LIN {X 0,Y 468.404,Z 515.595,A -85,B 0,C 180,E1 -7638.313,E2 -7638.313} C_VEL
LIN {X 0,Y 467.88,Z 524.784,A -85,B 0,C 180,E1 -7639.397,E2 -7639.397} C_VEL
LIN {X 0,Y 467.447,Z 533.686,A -85,B 0,C 180,E1 -7640.699,E2 -7640.699} C_VEL
LIN {X 0,Y 467.093,Z 540.848,A -85,B 0,C 180,E1 -7642,E2 -7642} C_VEL
LIN {X 0,Y 466.908,Z 547.07,A -85,B 0,C 180,E1 -7643.438,E2 -7643.438} C_VEL
LIN {X 0,Y 466.784,Z 551.676,A -85,B 0,C 180,E1 -7644.817,E2 -7644.817} C_VEL
LIN {X 0,Y 466.663,Z 553.957,A -85,B 0,C 180,E1 -7645.681,E2 -7645.681} C_VEL
LIN {X 0,Y 466.695,Z 555.806,A -85,B 0,C 180,E1 -7646.547,E2 -7646.547} C_VEL
LIN {X 0,Y 466.646,Z 557.193,A -85,B 0,C 180,E1 -7647.41,E2 -7647.41} C_VEL
LIN {X 0,Y 466.589,Z 558.785,A -85,B 0,C 180,E1 -7649.137,E2 -7649.137} C_VEL
LIN {X 0,Y 466.57,Z 559,A -85,B 0,C 180,E1 -7650,E2 -7650} C_VEL
LIN {X 0,Y 466.589,Z 558.786,A -85,B 0,C 180,E1 -7650.863,E2 -7650.863} C_VEL
LIN {X 0,Y 466.646,Z 557.196,A -85,B 0,C 180,E1 -7652.59,E2 -7652.59} C_VEL
LIN {X 0,Y 466.695,Z 555.81,A -85,B 0,C 180,E1 -7653.453,E2 -7653.453} C_VEL
LIN {X 0,Y 466.703,Z 552.895,A -85,B 0,C 180,E1 -7654.751,E2 -7654.751} C_VEL
LIN {X 0,Y 466.839,Z 548.948,A -85,B 0,C 180,E1 -7656.049,E2 -7656.049} C_VEL
LIN {X 0,Y 466.998,Z 542.875,A -85,B 0,C 180,E1 -7657.567,E2 -7657.567} C_VEL
LIN {X 0,Y 467.35,Z 536.235,A -85,B 0,C 180,E1 -7658.867,E2 -7658.867} C_VEL
LIN {X 0,Y 467.737,Z 527.992,A -85,B 0,C 180,E1 -7660.169,E2 -7660.169} C_VEL
LIN {X 0,Y 468.135,Z 519.518,A -85,B 0,C 180,E1 -7661.254,E2 -7661.254} C_VEL
LIN {X 0,Y 468.687,Z 509.169,A -85,B 0,C 180,E1 -7662.321,E2 -7662.321} C_VEL
LIN {X 0,Y 469.111,Z 497.566,A -85,B 0,C 180,E1 -7663.284,E2 -7663.284} C_VEL
LIN {X 0,Y 469.632,Z 485.232,A -85,B 0,C 180,E1 -7664.074,E2 -7664.074} C_VEL
LIN {X 0,Y 470.084,Z 472.858,A -85,B 0,C 180,E1 -7664.668,E2 -7664.668} C_VEL
LIN {X 0,Y 469.97,Z 467.485,A -85,B 0,C 180,E1 -7664.88,E2 -7664.88} C_VEL
LIN {X 0,Y 467.715,Z 454.277,A -85,B 0,C 180,E1 -7665.333,E2 -7665.333} C_VEL
LIN {X 0,Y 467.222,Z 450.988,A -85,B 0,C 180,E1 -7665.43,E2 -7665.43} C_VEL
LIN {X 0,Y 467.484,Z 441.099,A -85,B 0,C 180,E1 -7668.715,E2 -7668.715} C_VEL
LIN {X 0,Y 467.721,Z 432.418,A -85,B 0,C 180,E1 -7671.634,E2 -7671.634} C_VEL
LIN {X 0,Y 468.026,Z 423.02,A -85,B 0,C 180,E1 -7674.863,E2 -7674.863} C_VEL
LIN {X 0,Y 468.406,Z 414.945,A -85,B 0,C 180,E1 -7677.719,E2 -7677.719} C_VEL
LIN {X 0,Y 468.801,Z 405.09,A -85,B 0,C 180,E1 -7681.294,E2 -7681.294} C_VEL
LIN {X 0,Y 469.172,Z 397.613,A -85,B 0,C 180,E1 -7684.097,E2 -7684.097} C_VEL
LIN {X 0,Y 469.316,Z 392.645,A -85,B 0,C 180,E1 -7686.036,E2 -7686.036} C_VEL
LIN {X 0,Y 468.318,Z 386.339,A -85,B 0,C 180,E1 -7688.706,E2 -7688.706} C_VEL
LIN {X 0,Y 467.58,Z 382.245,A -85,B 0,C 180,E1 -7690.618,E2 -7690.618} C_VEL
LIN {X 0,Y 467.57,Z 382.25,A -85,B 0,C 180,E1 -7693.823,E2 -7693.823} C_VEL
LIN {X 0,Y 467.559,Z 382.242,A -85,B 0,C 180,E1 -7696.256,E2 -7696.256} C_VEL
LIN {X 0,Y 467.581,Z 382.242,A -85,B 0,C 180,E1 -7698.723,E2 -7698.723} C_VEL
LIN {X 0,Y 467.569,Z 382.242,A -85,B 0,C 180,E1 -7701.956,E2 -7701.956} C_VEL
LIN {X 0,Y 467.57,Z 382.244,A -85,B 0,C 180,E1 -7705.168,E2 -7705.168} C_VEL
LIN {X 0,Y 467.586,Z 382.24,A -85,B 0,C 180,E1 -7708.26,E2 -7708.26} C_VEL
LIN {X 0,Y 467.58,Z 382.24,A -85,B 0,C 180,E1 -7711.251,E2 -7711.251} C_VEL
LIN {X 0,Y 467.616,Z 382.236,A -85,B 0,C 180,E1 -7713.2,E2 -7713.2} C_VEL
LIN {X 0,Y 467.594,Z 382.241,A -85,B 0,C 180,E1 -7716.469,E2 -7716.469} C_VEL
LIN {X 0,Y 467.628,Z 382.235,A -85,B 0,C 180,E1 -7719.777,E2 -7719.777} C_VEL
LIN {X 0,Y 467.613,Z 382.238,A -85,B 0,C 180,E1 -7722.507,E2 -7722.507} C_VEL
LIN {X 0,Y 467.61,Z 382.235,A -85,B 0,C 180,E1 -7725.197,E2 -7725.197} C_VEL
LIN {X 0,Y 467.687,Z 382.228,A -85,B 0,C 180,E1 -7727.855,E2 -7727.855} C_VEL
LIN {X 0,Y 467.686,Z 382.228,A -85,B 0,C 180,E1 -7731.357,E2 -7731.357} C_VEL
LIN {X 0,Y 467.747,Z 382.22,A -85,B 0,C 180,E1 -7733.963,E2 -7733.963} C_VEL
LIN {X 0,Y 467.863,Z 382.203,A -85,B 0,C 180,E1 -7737.417,E2 -7737.417} C_VEL
LIN {X 0,Y 467.887,Z 382.205,A -85,B 0,C 180,E1 -7740,E2 -7740} C_VEL
LIN {X 0,Y 467.862,Z 382.206,A -85,B 0,C 180,E1 -7742.583,E2 -7742.583} C_VEL
LIN {X 0,Y 467.748,Z 382.22,A -85,B 0,C 180,E1 -7746.037,E2 -7746.037} C_VEL
LIN {X 0,Y 467.683,Z 382.229,A -85,B 0,C 180,E1 -7748.643,E2 -7748.643} C_VEL
LIN {X 0,Y 467.66,Z 382.234,A -85,B 0,C 180,E1 -7752.145,E2 -7752.145} C_VEL
LIN {X 0,Y 467.643,Z 382.236,A -85,B 0,C 180,E1 -7755.695,E2 -7755.695} C_VEL
LIN {X 0,Y 467.627,Z 382.235,A -85,B 0,C 180,E1 -7759.308,E2 -7759.308} C_VEL
LIN {X 0,Y 467.538,Z 382.25,A -85,B 0,C 180,E1 -7762.074,E2 -7762.074} C_VEL
LIN {X 0,Y 467.589,Z 382.238,A -85,B 0,C 180,E1 -7764.888,E2 -7764.888} C_VEL
LIN {X 0,Y 467.631,Z 382.236,A -85,B 0,C 180,E1 -7767.768,E2 -7767.768} C_VEL
LIN {X 0,Y 467.571,Z 382.242,A -85,B 0,C 180,E1 -7771.045,E2 -7771.045} C_VEL
LIN {X 0,Y 467.592,Z 382.241,A -85,B 0,C 180,E1 -7774.242,E2 -7774.242} C_VEL
LIN {X 0,Y 467.551,Z 382.243,A -85,B 0,C 180,E1 -7777.186,E2 -7777.186} C_VEL
LIN {X 0,Y 467.581,Z 382.241,A -85,B 0,C 180,E1 -7780.265,E2 -7780.265} C_VEL
LIN {X 0,Y 467.589,Z 382.24,A -85,B 0,C 180,E1 -7782.567,E2 -7782.567} C_VEL
LIN {X 0,Y 467.575,Z 382.242,A -85,B 0,C 180,E1 -7786.177,E2 -7786.177} C_VEL
LIN {X 0,Y 467.587,Z 382.237,A -85,B 0,C 180,E1 -7788.722,E2 -7788.722} C_VEL
LIN {X 0,Y 467.564,Z 382.243,A -85,B 0,C 180,E1 -7791.955,E2 -7791.955} C_VEL
LIN {X 0,Y 467.434,Z 382.262,A -85,B 0,C 180,E1 -7795.156,E2 -7795.156} C_VEL
LIN {X 0,Y 467.22,Z 382.29,A -85,B 0,C 180,E1 -7797.391,E2 -7797.391} C_VEL
LIN {X 0,Y 467.124,Z 382.618,A -85,B 0,C 180,E1 -7798.225,E2 -7798.225} C_VEL
LIN {X 0,Y 467.082,Z 385.538,A -85,B 0,C 180,E1 -7801.217,E2 -7801.217} C_VEL
LIN {X 0,Y 467.017,Z 388.795,A -85,B 0,C 180,E1 -7804.545,E2 -7804.545} C_VEL
LIN {X 0,Y 466.878,Z 392.162,A -85,B 0,C 180,E1 -7807.893,E2 -7807.893} C_VEL
LIN {X 0,Y 466.856,Z 395.11,A -85,B 0,C 180,E1 -7810.659,E2 -7810.659} C_VEL
LIN {X 0,Y 466.821,Z 398.837,A -85,B 0,C 180,E1 -7813.93,E2 -7813.93} C_VEL
LIN {X 0,Y 466.77,Z 399.842,A -85,B 0,C 180,E1 -7814.23,E2 -7814.23} C_VEL
LIN {X 0,Y 466.543,Z 402.574,A -85,B 0,C 180,E1 -7814.555,E2 -7814.555} C_VEL
LIN {X 0,Y 466.119,Z 406.733,A -85,B 0,C 180,E1 -7814.803,E2 -7814.803} C_VEL
LIN {X 0,Y 463.509,Z 424.033,A -85,B 0,C 180,E1 -7815.447,E2 -7815.447} C_VEL
LIN {X 0,Y 463.214,Z 427.363,A -85,B 0,C 180,E1 -7815.614,E2 -7815.614} C_VEL
LIN {X 0,Y 462.772,Z 438.749,A -85,B 0,C 180,E1 -7816.313,E2 -7816.313} C_VEL
LIN {X 0,Y 462.312,Z 449.522,A -85,B 0,C 180,E1 -7817.154,E2 -7817.154} C_VEL
LIN {X 0,Y 461.81,Z 459.725,A -85,B 0,C 180,E1 -7818.144,E2 -7818.144} C_VEL
LIN {X 0,Y 461.272,Z 468.878,A -85,B 0,C 180,E1 -7819.243,E2 -7819.243} C_VEL
LIN {X 0,Y 460.84,Z 477.749,A -85,B 0,C 180,E1 -7820.564,E2 -7820.564} C_VEL
LIN {X 0,Y 460.394,Z 484.894,A -85,B 0,C 180,E1 -7821.883,E2 -7821.883} C_VEL
LIN {X 0,Y 460.123,Z 490.324,A -85,B 0,C 180,E1 -7823.133,E2 -7823.133} C_VEL
LIN {X 0,Y 459.892,Z 494.386,A -85,B 0,C 180,E1 -7824.299,E2 -7824.299} C_VEL
LIN {X 0,Y 459.881,Z 497.956,A -85,B 0,C 180,E1 -7825.618,E2 -7825.618} C_VEL
LIN {X 0,Y 459.779,Z 499.808,A -85,B 0,C 180,E1 -7826.495,E2 -7826.495} C_VEL
LIN {X 0,Y 459.768,Z 501.199,A -85,B 0,C 180,E1 -7827.372,E2 -7827.372} C_VEL
LIN {X 0,Y 459.557,Z 502.809,A -85,B 0,C 180,E1 -7829.124,E2 -7829.124} C_VEL
LIN {X 0,Y 459.536,Z 503.043,A -85,B 0,C 180,E1 -7830,E2 -7830} C_VEL
LIN {X 0,Y 459.639,Z 502.274,A -85,B 0,C 180,E1 -7831.753,E2 -7831.753} C_VEL
LIN {X 0,Y 459.768,Z 501.31,A -85,B 0,C 180,E1 -7832.628,E2 -7832.628} C_VEL
LIN {X 0,Y 459.78,Z 499.967,A -85,B 0,C 180,E1 -7833.505,E2 -7833.505} C_VEL
LIN {X 0,Y 459.846,Z 497.126,A -85,B 0,C 180,E1 -7834.822,E2 -7834.822} C_VEL
LIN {X 0,Y 460.021,Z 493.267,A -85,B 0,C 180,E1 -7836.139,E2 -7836.139} C_VEL
LIN {X 0,Y 460.196,Z 488.291,A -85,B 0,C 180,E1 -7837.459,E2 -7837.459} C_VEL
LIN {X 0,Y 460.571,Z 482.016,A -85,B 0,C 180,E1 -7838.777,E2 -7838.777} C_VEL
LIN {X 0,Y 460.971,Z 474.16,A -85,B 0,C 180,E1 -7840.098,E2 -7840.098} C_VEL
LIN {X 0,Y 461.518,Z 464.377,A -85,B 0,C 180,E1 -7841.418,E2 -7841.418} C_VEL
LIN {X 0,Y 462.073,Z 454.105,A -85,B 0,C 180,E1 -7842.518,E2 -7842.518} C_VEL
LIN {X 0,Y 462.528,Z 442.951,A -85,B 0,C 180,E1 -7843.476,E2 -7843.476} C_VEL
LIN {X 0,Y 463.071,Z 430.963,A -85,B 0,C 180,E1 -7844.278,E2 -7844.278} C_VEL
LIN {X 0,Y 463.458,Z 418.943,A -85,B 0,C 180,E1 -7844.883,E2 -7844.883} C_VEL
LIN {X 0,Y 463.495,Z 415.951,A -85,B 0,C 180,E1 -7845.012,E2 -7845.012} C_VEL
LIN {X 0,Y 460.557,Z 403.288,A -85,B 0,C 180,E1 -7845.535,E2 -7845.535} C_VEL
LIN {X 0,Y 459.806,Z 400.064,A -85,B 0,C 180,E1 -7845.667,E2 -7845.667} C_VEL
LIN {X 0,Y 459.784,Z 396.594,A -85,B 0,C 180,E1 -7848.723,E2 -7848.723} C_VEL
LIN {X 0,Y 459.828,Z 393.59,A -85,B 0,C 180,E1 -7851.52,E2 -7851.52} C_VEL
LIN {X 0,Y 459.896,Z 390.686,A -85,B 0,C 180,E1 -7854.369,E2 -7854.369} C_VEL
LIN {X 0,Y 459.989,Z 387.461,A -85,B 0,C 180,E1 -7857.605,E2 -7857.605} C_VEL
LIN {X 0,Y 460.056,Z 384.906,A -85,B 0,C 180,E1 -7860.273,E2 -7860.273} C_VEL
LIN {X 0,Y 460.108,Z 383.174,A -85,B 0,C 180,E1 -7862.318,E2 -7862.318} C_VEL
LIN {X 0,Y 460.434,Z 383.131,A -85,B 0,C 180,E1 -7865.453,E2 -7865.453} C_VEL
LIN {X 0,Y 460.548,Z 383.118,A -85,B 0,C 180,E1 -7868.898,E2 -7868.898} C_VEL
LIN {X 0,Y 460.527,Z 383.121,A -85,B 0,C 180,E1 -7872.181,E2 -7872.181} C_VEL
LIN {X 0,Y 460.517,Z 383.12,A -85,B 0,C 180,E1 -7875.411,E2 -7875.411} C_VEL
LIN {X 0,Y 460.536,Z 383.119,A -85,B 0,C 180,E1 -7878.398,E2 -7878.398} C_VEL
LIN {X 0,Y 460.531,Z 383.118,A -85,B 0,C 180,E1 -7881.267,E2 -7881.267} C_VEL
LIN {X 0,Y 460.517,Z 383.121,A -85,B 0,C 180,E1 -7884.555,E2 -7884.555} C_VEL
LIN {X 0,Y 460.536,Z 383.12,A -85,B 0,C 180,E1 -7887.716,E2 -7887.716} C_VEL
LIN {X 0,Y 460.545,Z 383.118,A -85,B 0,C 180,E1 -7890.769,E2 -7890.769} C_VEL
LIN {X 0,Y 460.56,Z 383.115,A -85,B 0,C 180,E1 -7893.734,E2 -7893.734} C_VEL
LIN {X 0,Y 460.549,Z 383.115,A -85,B 0,C 180,E1 -7896.624,E2 -7896.624} C_VEL
LIN {X 0,Y 460.557,Z 383.116,A -85,B 0,C 180,E1 -7899.453,E2 -7899.453} C_VEL
LIN {X 0,Y 460.555,Z 383.117,A -85,B 0,C 180,E1 -7902.23,E2 -7902.23} C_VEL
LIN {X 0,Y 460.571,Z 383.114,A -85,B 0,C 180,E1 -7904.965,E2 -7904.965} C_VEL
LIN {X 0,Y 460.616,Z 383.107,A -85,B 0,C 180,E1 -7908.559,E2 -7908.559} C_VEL
LIN {X 0,Y 460.625,Z 383.106,A -85,B 0,C 180,E1 -7911.224,E2 -7911.224} C_VEL
LIN {X 0,Y 460.712,Z 383.097,A -85,B 0,C 180,E1 -7913.87,E2 -7913.87} C_VEL
LIN {X 0,Y 460.804,Z 383.086,A -85,B 0,C 180,E1 -7917.377,E2 -7917.377} C_VEL
LIN {X 0,Y 460.858,Z 383.081,A -85,B 0,C 180,E1 -7920,E2 -7920} C_VEL
LIN {X 0,Y 460.805,Z 383.082,A -85,B 0,C 180,E1 -7922.622,E2 -7922.622} C_VEL
LIN {X 0,Y 460.715,Z 383.096,A -85,B 0,C 180,E1 -7926.13,E2 -7926.13} C_VEL
LIN {X 0,Y 460.634,Z 383.106,A -85,B 0,C 180,E1 -7928.776,E2 -7928.776} C_VEL
LIN {X 0,Y 460.639,Z 383.105,A -85,B 0,C 180,E1 -7932.457,E2 -7932.457} C_VEL
LIN {X 0,Y 460.605,Z 383.108,A -85,B 0,C 180,E1 -7935.997,E2 -7935.997} C_VEL
LIN {X 0,Y 460.574,Z 383.114,A -85,B 0,C 180,E1 -7939.615,E2 -7939.615} C_VEL
LIN {X 0,Y 460.515,Z 383.121,A -85,B 0,C 180,E1 -7942.428,E2 -7942.428} C_VEL
LIN {X 0,Y 460.557,Z 383.117,A -85,B 0,C 180,E1 -7945.798,E2 -7945.798} C_VEL
LIN {X 0,Y 460.56,Z 383.113,A -85,B 0,C 180,E1 -7948.233,E2 -7948.233} C_VEL
LIN {X 0,Y 460.525,Z 383.121,A -85,B 0,C 180,E1 -7951.283,E2 -7951.283} C_VEL
LIN {X 0,Y 460.536,Z 383.119,A -85,B 0,C 180,E1 -7954.505,E2 -7954.505} C_VEL
LIN {X 0,Y 460.505,Z 383.124,A -85,B 0,C 180,E1 -7957.623,E2 -7957.623} C_VEL
LIN {X 0,Y 460.545,Z 383.116,A -85,B 0,C 180,E1 -7960.269,E2 -7960.269} C_VEL
LIN {X 0,Y 460.504,Z 383.125,A -85,B 0,C 180,E1 -7963.375,E2 -7963.375} C_VEL
LIN {X 0,Y 460.512,Z 383.123,A -85,B 0,C 180,E1 -7966.626,E2 -7966.626} C_VEL
LIN {X 0,Y 460.571,Z 383.226,A -85,B 0,C 180,E1 -7969.188,E2 -7969.188} C_VEL
LIN {X 0,Y 461.891,Z 390.612,A -85,B 0,C 180,E1 -7972.509,E2 -7972.509} C_VEL
LIN {X 0,Y 462.366,Z 394.643,A -85,B 0,C 180,E1 -7974.206,E2 -7974.206} C_VEL
LIN {X 0,Y 461.99,Z 402.601,A -85,B 0,C 180,E1 -7977.313,E2 -7977.313} C_VEL
LIN {X 0,Y 461.572,Z 410.362,A -85,B 0,C 180,E1 -7980.215,E2 -7980.215} C_VEL
LIN {X 0,Y 461.217,Z 418.825,A -85,B 0,C 180,E1 -7983.287,E2 -7983.287} C_VEL
LIN {X 0,Y 460.863,Z 426.994,A -85,B 0,C 180,E1 -7986.203,E2 -7986.203} C_VEL
LIN {X 0,Y 460.613,Z 435.003,A -85,B 0,C 180,E1 -7988.994,E2 -7988.994} C_VEL
LIN {X 0,Y 460.37,Z 443.128,A -85,B 0,C 180,E1 -7991.763,E2 -7991.763} C_VEL
LIN {X 0,Y 460.167,Z 450.705,A -85,B 0,C 180,E1 -7994.337,E2 -7994.337} C_VEL
LIN {X 0,Y 462.581,Z 465.278,A -85,B 0,C 180,E1 -7994.812,E2 -7994.812} C_VEL
LIN {X 0,Y 463.264,Z 471.127,A -85,B 0,C 180,E1 -7995.054,E2 -7995.054} C_VEL
LIN {X 0,Y 462.835,Z 482.805,A -85,B 0,C 180,E1 -7995.602,E2 -7995.602} C_VEL
LIN {X 0,Y 462.286,Z 495.149,A -85,B 0,C 180,E1 -7996.37,E2 -7996.37} C_VEL
LIN {X 0,Y 461.877,Z 505.147,A -85,B 0,C 180,E1 -7997.162,E2 -7997.162} C_VEL
LIN {X 0,Y 461.399,Z 515.159,A -85,B 0,C 180,E1 -7998.133,E2 -7998.133} C_VEL
LIN {X 0,Y 460.865,Z 524.377,A -85,B 0,C 180,E1 -7999.233,E2 -7999.233} C_VEL
LIN {X 0,Y 460.418,Z 533.368,A -85,B 0,C 180,E1 -8000.555,E2 -8000.555} C_VEL
LIN {X 0,Y 460.055,Z 540.609,A -85,B 0,C 180,E1 -8001.876,E2 -8001.876} C_VEL
LIN {X 0,Y 459.848,Z 545.5,A -85,B 0,C 180,E1 -8002.977,E2 -8002.977} C_VEL
LIN {X 0,Y 459.756,Z 550.262,A -85,B 0,C 180,E1 -8004.297,E2 -8004.297} C_VEL
LIN {X 0,Y 459.579,Z 553.894,A -85,B 0,C 180,E1 -8005.615,E2 -8005.615} C_VEL
LIN {X 0,Y 459.591,Z 555.773,A -85,B 0,C 180,E1 -8006.493,E2 -8006.493} C_VEL
LIN {X 0,Y 459.57,Z 557.175,A -85,B 0,C 180,E1 -8007.37,E2 -8007.37} C_VEL
LIN {X 0,Y 459.494,Z 558.779,A -85,B 0,C 180,E1 -8009.124,E2 -8009.124} C_VEL
LIN {X 0,Y 459.474,Z 558.994,A -85,B 0,C 180,E1 -8010,E2 -8010} C_VEL
LIN {X 0,Y 459.494,Z 558.779,A -85,B 0,C 180,E1 -8010.876,E2 -8010.876} C_VEL
LIN {X 0,Y 459.57,Z 557.178,A -85,B 0,C 180,E1 -8012.629,E2 -8012.629} C_VEL
LIN {X 0,Y 459.591,Z 555.777,A -85,B 0,C 180,E1 -8013.507,E2 -8013.507} C_VEL
LIN {X 0,Y 459.634,Z 552.818,A -85,B 0,C 180,E1 -8014.824,E2 -8014.824} C_VEL
LIN {X 0,Y 459.757,Z 548.815,A -85,B 0,C 180,E1 -8016.143,E2 -8016.143} C_VEL
LIN {X 0,Y 459.929,Z 542.66,A -85,B 0,C 180,E1 -8017.684,E2 -8017.684} C_VEL
LIN {X 0,Y 460.287,Z 535.945,A -85,B 0,C 180,E1 -8019.004,E2 -8019.004} C_VEL
LIN {X 0,Y 460.7,Z 527.616,A -85,B 0,C 180,E1 -8020.326,E2 -8020.326} C_VEL
LIN {X 0,Y 461.146,Z 519.085,A -85,B 0,C 180,E1 -8021.427,E2 -8021.427} C_VEL
LIN {X 0,Y 461.697,Z 508.871,A -85,B 0,C 180,E1 -8022.498,E2 -8022.498} C_VEL
LIN {X 0,Y 462.119,Z 498.133,A -85,B 0,C 180,E1 -8023.41,E2 -8023.41} C_VEL
LIN {X 0,Y 462.643,Z 486.726,A -85,B 0,C 180,E1 -8024.179,E2 -8024.179} C_VEL
LIN {X 0,Y 463.147,Z 475.036,A -85,B 0,C 180,E1 -8024.781,E2 -8024.781} C_VEL
LIN {X 0,Y 463.102,Z 468.615,A -85,B 0,C 180,E1 -8025.048,E2 -8025.048} C_VEL
LIN {X 0,Y 460.884,Z 455.323,A -85,B 0,C 180,E1 -8025.529,E2 -8025.529} C_VEL
LIN {X 0,Y 460.148,Z 450.492,A -85,B 0,C 180,E1 -8025.689,E2 -8025.689} C_VEL
LIN {X 0,Y 460.454,Z 440.268,A -85,B 0,C 180,E1 -8029.178,E2 -8029.178} C_VEL
LIN {X 0,Y 460.728,Z 430.871,A -85,B 0,C 180,E1 -8032.418,E2 -8032.418} C_VEL
LIN {X 0,Y 461.117,Z 420.914,A -85,B 0,C 180,E1 -8035.942,E2 -8035.942} C_VEL
LIN {X 0,Y 461.43,Z 413.371,A -85,B 0,C 180,E1 -8038.671,E2 -8038.671} C_VEL
LIN {X 0,Y 461.828,Z 405.593,A -85,B 0,C 180,E1 -8041.548,E2 -8041.548} C_VEL
LIN {X 0,Y 462.191,Z 398.56,A -85,B 0,C 180,E1 -8044.237,E2 -8044.237} C_VEL
LIN {X 0,Y 462.263,Z 393.36,A -85,B 0,C 180,E1 -8046.314,E2 -8046.314} C_VEL
LIN {X 0,Y 461.257,Z 387.152,A -85,B 0,C 180,E1 -8049.007,E2 -8049.007} C_VEL
LIN {X 0,Y 460.553,Z 383.12,A -85,B 0,C 180,E1 -8050.911,E2 -8050.911} C_VEL
LIN {X 0,Y 460.522,Z 383.128,A -85,B 0,C 180,E1 -8054.171,E2 -8054.171} C_VEL
LIN {X 0,Y 460.516,Z 383.125,A -85,B 0,C 180,E1 -8057.1,E2 -8057.1} C_VEL
LIN {X 0,Y 460.561,Z 383.117,A -85,B 0,C 180,E1 -8060.14,E2 -8060.14} C_VEL
LIN {X 0,Y 460.481,Z 383.127,A -85,B 0,C 180,E1 -8063.471,E2 -8063.471} C_VEL
LIN {X 0,Y 460.532,Z 383.119,A -85,B 0,C 180,E1 -8066.675,E2 -8066.675} C_VEL
LIN {X 0,Y 460.514,Z 383.119,A -85,B 0,C 180,E1 -8069.76,E2 -8069.76} C_VEL
LIN {X 0,Y 460.581,Z 383.115,A -85,B 0,C 180,E1 -8072.757,E2 -8072.757} C_VEL
LIN {X 0,Y 460.534,Z 383.118,A -85,B 0,C 180,E1 -8075.667,E2 -8075.667} C_VEL
LIN {X 0,Y 460.525,Z 383.121,A -85,B 0,C 180,E1 -8078.578,E2 -8078.578} C_VEL
LIN {X 0,Y 460.595,Z 383.111,A -85,B 0,C 180,E1 -8081.311,E2 -8081.311} C_VEL
LIN {X 0,Y 460.607,Z 383.108,A -85,B 0,C 180,E1 -8084.059,E2 -8084.059} C_VEL
LIN {X 0,Y 460.634,Z 383.105,A -85,B 0,C 180,E1 -8087.667,E2 -8087.667} C_VEL
LIN {X 0,Y 460.633,Z 383.107,A -85,B 0,C 180,E1 -8091.224,E2 -8091.224} C_VEL
LIN {X 0,Y 460.713,Z 383.096,A -85,B 0,C 180,E1 -8093.87,E2 -8093.87} C_VEL
LIN {X 0,Y 460.804,Z 383.082,A -85,B 0,C 180,E1 -8097.378,E2 -8097.378} C_VEL
LIN {X 0,Y 460.857,Z 383.08,A -85,B 0,C 180,E1 -8100,E2 -8100} C_VEL
LIN {X 0,Y 460.803,Z 383.086,A -85,B 0,C 180,E1 -8102.623,E2 -8102.623} C_VEL
LIN {X 0,Y 460.714,Z 383.097,A -85,B 0,C 180,E1 -8106.13,E2 -8106.13} C_VEL
LIN {X 0,Y 460.631,Z 383.106,A -85,B 0,C 180,E1 -8108.776,E2 -8108.776} C_VEL
LIN {X 0,Y 460.617,Z 383.108,A -85,B 0,C 180,E1 -8112.445,E2 -8112.445} C_VEL
LIN {X 0,Y 460.604,Z 383.111,A -85,B 0,C 180,E1 -8115.998,E2 -8115.998} C_VEL
LIN {X 0,Y 460.573,Z 383.114,A -85,B 0,C 180,E1 -8119.615,E2 -8119.615} C_VEL
LIN {X 0,Y 460.514,Z 383.121,A -85,B 0,C 180,E1 -8122.429,E2 -8122.429} C_VEL
LIN {X 0,Y 460.556,Z 383.119,A -85,B 0,C 180,E1 -8125.798,E2 -8125.798} C_VEL
LIN {X 0,Y 460.559,Z 383.116,A -85,B 0,C 180,E1 -8128.233,E2 -8128.233} C_VEL
LIN {X 0,Y 460.524,Z 383.121,A -85,B 0,C 180,E1 -8131.283,E2 -8131.283} C_VEL
LIN {X 0,Y 460.535,Z 383.117,A -85,B 0,C 180,E1 -8134.506,E2 -8134.506} C_VEL
LIN {X 0,Y 460.531,Z 383.122,A -85,B 0,C 180,E1 -8137.621,E2 -8137.621} C_VEL
LIN {X 0,Y 460.545,Z 383.118,A -85,B 0,C 180,E1 -8140.269,E2 -8140.269} C_VEL
LIN {X 0,Y 460.499,Z 383.124,A -85,B 0,C 180,E1 -8143.376,E2 -8143.376} C_VEL
LIN {X 0,Y 460.526,Z 383.118,A -85,B 0,C 180,E1 -8146.627,E2 -8146.627} C_VEL
LIN {X 0,Y 460.546,Z 383.119,A -85,B 0,C 180,E1 -8149.73,E2 -8149.73} C_VEL
LIN {X 0,Y 460.498,Z 383.122,A -85,B 0,C 180,E1 -8152.525,E2 -8152.525} C_VEL
LIN {X 0,Y 460.357,Z 383.145,A -85,B 0,C 180,E1 -8155.608,E2 -8155.608} C_VEL
LIN {X 0,Y 460.117,Z 383.174,A -85,B 0,C 180,E1 -8157.683,E2 -8157.683} C_VEL
LIN {X 0,Y 460.04,Z 384.846,A -85,B 0,C 180,E1 -8159.726,E2 -8159.726} C_VEL
LIN {X 0,Y 459.98,Z 387.737,A -85,B 0,C 180,E1 -8162.718,E2 -8162.718} C_VEL
LIN {X 0,Y 459.905,Z 390.598,A -85,B 0,C 180,E1 -8165.632,E2 -8165.632} C_VEL
LIN {X 0,Y 459.821,Z 393.82,A -85,B 0,C 180,E1 -8168.803,E2 -8168.803} C_VEL
LIN {X 0,Y 459.792,Z 397.505,A -85,B 0,C 180,E1 -8172.199,E2 -8172.199} C_VEL
LIN {X 0,Y 459.796,Z 400.147,A -85,B 0,C 180,E1 -8174.45,E2 -8174.45} C_VEL
LIN {X 0,Y 462.964,Z 413.491,A -85,B 0,C 180,E1 -8174.968,E2 -8174.968} C_VEL
LIN {X 0,Y 463.514,Z 416.83,A -85,B 0,C 180,E1 -8175.119,E2 -8175.119} C_VEL
LIN {X 0,Y 463.214,Z 427.363,A -85,B 0,C 180,E1 -8175.614,E2 -8175.614} C_VEL
LIN {X 0,Y 462.367,Z 432.81,A -85,B 0,C 180,E1 -8175.903,E2 -8175.903} C_VEL
LIN {X 0,Y 459.267,Z 441.437,A -85,B 0,C 180,E1 -8176.384,E2 -8176.384} C_VEL
LIN {X 0,Y 456.107,Z 449.62,A -85,B 0,C 180,E1 -8176.948,E2 -8176.948} C_VEL
LIN {X 0,Y 455.164,Z 454.344,A -85,B 0,C 180,E1 -8177.363,E2 -8177.363} C_VEL
LIN {X 0,Y 454.589,Z 464.053,A -85,B 0,C 180,E1 -8178.406,E2 -8178.406} C_VEL
LIN {X 0,Y 454.142,Z 472.517,A -85,B 0,C 180,E1 -8179.523,E2 -8179.523} C_VEL
LIN {X 0,Y 453.677,Z 480.733,A -85,B 0,C 180,E1 -8180.864,E2 -8180.864} C_VEL
LIN {X 0,Y 453.339,Z 486.353,A -85,B 0,C 180,E1 -8181.98,E2 -8181.98} C_VEL
LIN {X 0,Y 453.083,Z 492.103,A -85,B 0,C 180,E1 -8183.398,E2 -8183.398} C_VEL
LIN {X 0,Y 452.724,Z 496.129,A -85,B 0,C 180,E1 -8184.656,E2 -8184.656} C_VEL
LIN {X 0,Y 452.809,Z 498.39,A -85,B 0,C 180,E1 -8185.549,E2 -8185.549} C_VEL
LIN {X 0,Y 452.718,Z 500.239,A -85,B 0,C 180,E1 -8186.44,E2 -8186.44} C_VEL
LIN {X 0,Y 452.697,Z 501.63,A -85,B 0,C 180,E1 -8187.331,E2 -8187.331} C_VEL
LIN {X 0,Y 452.493,Z 503.239,A -85,B 0,C 180,E1 -8189.11,E2 -8189.11} C_VEL
LIN {X 0,Y 452.47,Z 503.474,A -85,B 0,C 180,E1 -8190,E2 -8190} C_VEL
LIN {X 0,Y 452.58,Z 502.704,A -85,B 0,C 180,E1 -8191.78,E2 -8191.78} C_VEL
LIN {X 0,Y 452.683,Z 501.741,A -85,B 0,C 180,E1 -8192.67,E2 -8192.67} C_VEL
LIN {X 0,Y 452.718,Z 500.397,A -85,B 0,C 180,E1 -8193.56,E2 -8193.56} C_VEL
LIN {X 0,Y 452.772,Z 497.557,A -85,B 0,C 180,E1 -8194.898,E2 -8194.898} C_VEL
LIN {X 0,Y 452.986,Z 493.697,A -85,B 0,C 180,E1 -8196.235,E2 -8196.235} C_VEL
LIN {X 0,Y 453.163,Z 488.721,A -85,B 0,C 180,E1 -8197.575,E2 -8197.575} C_VEL
LIN {X 0,Y 453.556,Z 482.446,A -85,B 0,C 180,E1 -8198.914,E2 -8198.914} C_VEL
LIN {X 0,Y 454.007,Z 474.587,A -85,B 0,C 180,E1 -8200.255,E2 -8200.255} C_VEL
LIN {X 0,Y 454.572,Z 464.805,A -85,B 0,C 180,E1 -8201.595,E2 -8201.595} C_VEL
LIN {X 0,Y 455.175,Z 454.531,A -85,B 0,C 180,E1 -8202.711,E2 -8202.711} C_VEL
LIN {X 0,Y 455.637,Z 443.785,A -85,B 0,C 180,E1 -8203.651,E2 -8203.651} C_VEL
LIN {X 0,Y 456.131,Z 433.207,A -85,B 0,C 180,E1 -8204.386,E2 -8204.386} C_VEL
LIN {X 0,Y 456.573,Z 420.659,A -85,B 0,C 180,E1 -8205.056,E2 -8205.056} C_VEL
LIN {X 0,Y 456.552,Z 416.652,A -85,B 0,C 180,E1 -8205.233,E2 -8205.233} C_VEL
LIN {X 0,Y 453.59,Z 404.1,A -85,B 0,C 180,E1 -8205.77,E2 -8205.77} C_VEL
LIN {X 0,Y 452.716,Z 400.49,A -85,B 0,C 180,E1 -8205.905,E2 -8205.905} C_VEL
LIN {X 0,Y 452.711,Z 396.973,A -85,B 0,C 180,E1 -8209.027,E2 -8209.027} C_VEL
LIN {X 0,Y 452.769,Z 393.937,A -85,B 0,C 180,E1 -8211.872,E2 -8211.872} C_VEL
LIN {X 0,Y 452.86,Z 391.004,A -85,B 0,C 180,E1 -8214.773,E2 -8214.773} C_VEL
LIN {X 0,Y 452.935,Z 387.994,A -85,B 0,C 180,E1 -8217.816,E2 -8217.816} C_VEL
LIN {X 0,Y 452.992,Z 385.147,A -85,B 0,C 180,E1 -8220.796,E2 -8220.796} C_VEL
LIN {X 0,Y 453.008,Z 384.169,A -85,B 0,C 180,E1 -8221.836,E2 -8221.836} C_VEL
LIN {X 0,Y 453.364,Z 384.014,A -85,B 0,C 180,E1 -8225,E2 -8225} C_VEL
LIN {X 0,Y 453.466,Z 384,A -85,B 0,C 180,E1 -8228.312,E2 -8228.312} C_VEL
LIN {X 0,Y 453.498,Z 383.997,A -85,B 0,C 180,E1 -8230.609,E2 -8230.609} C_VEL
LIN {X 0,Y 453.458,Z 383.999,A -85,B 0,C 180,E1 -8233.244,E2 -8233.244} C_VEL
LIN {X 0,Y 453.466,Z 384,A -85,B 0,C 180,E1 -8235.779,E2 -8235.779} C_VEL
LIN {X 0,Y 453.483,Z 383.998,A -85,B 0,C 180,E1 -8238.209,E2 -8238.209} C_VEL
LIN {X 0,Y 453.52,Z 383.993,A -85,B 0,C 180,E1 -8240.79,E2 -8240.79} C_VEL
LIN {X 0,Y 453.461,Z 384,A -85,B 0,C 180,E1 -8243.918,E2 -8243.918} C_VEL
LIN {X 0,Y 453.487,Z 383.995,A -85,B 0,C 180,E1 -8247.151,E2 -8247.151} C_VEL
LIN {X 0,Y 453.48,Z 383.998,A -85,B 0,C 180,E1 -8250.268,E2 -8250.268} C_VEL
LIN {X 0,Y 453.506,Z 383.993,A -85,B 0,C 180,E1 -8253.294,E2 -8253.294} C_VEL
LIN {X 0,Y 453.503,Z 383.997,A -85,B 0,C 180,E1 -8256.239,E2 -8256.239} C_VEL
LIN {X 0,Y 453.488,Z 383.995,A -85,B 0,C 180,E1 -8259.118,E2 -8259.118} C_VEL
LIN {X 0,Y 453.509,Z 383.995,A -85,B 0,C 180,E1 -8261.944,E2 -8261.944} C_VEL
LIN {X 0,Y 453.545,Z 383.989,A -85,B 0,C 180,E1 -8264.726,E2 -8264.726} C_VEL
LIN {X 0,Y 453.564,Z 383.986,A -85,B 0,C 180,E1 -8268.379,E2 -8268.379} C_VEL
LIN {X 0,Y 453.59,Z 383.982,A -85,B 0,C 180,E1 -8271.087,E2 -8271.087} C_VEL
LIN {X 0,Y 453.678,Z 383.974,A -85,B 0,C 180,E1 -8273.775,E2 -8273.775} C_VEL
LIN {X 0,Y 453.748,Z 383.965,A -85,B 0,C 180,E1 -8277.337,E2 -8277.337} C_VEL
LIN {X 0,Y 453.828,Z 383.956,A -85,B 0,C 180,E1 -8280,E2 -8280} C_VEL
LIN {X 0,Y 453.749,Z 383.961,A -85,B 0,C 180,E1 -8282.663,E2 -8282.663} C_VEL
LIN {X 0,Y 453.682,Z 383.972,A -85,B 0,C 180,E1 -8286.225,E2 -8286.225} C_VEL
LIN {X 0,Y 453.598,Z 383.983,A -85,B 0,C 180,E1 -8288.913,E2 -8288.913} C_VEL
LIN {X 0,Y 453.607,Z 383.98,A -85,B 0,C 180,E1 -8292.551,E2 -8292.551} C_VEL
LIN {X 0,Y 453.549,Z 383.986,A -85,B 0,C 180,E1 -8296.196,E2 -8296.196} C_VEL
LIN {X 0,Y 453.523,Z 383.994,A -85,B 0,C 180,E1 -8299.04,E2 -8299.04} C_VEL
LIN {X 0,Y 453.481,Z 383.999,A -85,B 0,C 180,E1 -8301.836,E2 -8301.836} C_VEL
LIN {X 0,Y 453.505,Z 383.995,A -85,B 0,C 180,E1 -8304.735,E2 -8304.735} C_VEL
LIN {X 0,Y 453.542,Z 383.988,A -85,B 0,C 180,E1 -8307.961,E2 -8307.961} C_VEL
LIN {X 0,Y 453.47,Z 383.999,A -85,B 0,C 180,E1 -8311.525,E2 -8311.525} C_VEL
LIN {X 0,Y 453.491,Z 383.998,A -85,B 0,C 180,E1 -8314.777,E2 -8314.777} C_VEL
LIN {X 0,Y 453.468,Z 383.998,A -85,B 0,C 180,E1 -8318.311,E2 -8318.311} C_VEL
LIN {X 0,Y 453.497,Z 383.994,A -85,B 0,C 180,E1 -8320.609,E2 -8320.609} C_VEL
LIN {X 0,Y 453.46,Z 384.003,A -85,B 0,C 180,E1 -8323.244,E2 -8323.244} C_VEL
LIN {X 0,Y 453.477,Z 383.998,A -85,B 0,C 180,E1 -8325.78,E2 -8325.78} C_VEL
LIN {X 0,Y 453.541,Z 384.134,A -85,B 0,C 180,E1 -8328.89,E2 -8328.89} C_VEL
LIN {X 0,Y 454.948,Z 392.015,A -85,B 0,C 180,E1 -8332.496,E2 -8332.496} C_VEL
LIN {X 0,Y 455.374,Z 395.743,A -85,B 0,C 180,E1 -8334.093,E2 -8334.093} C_VEL
LIN {X 0,Y 455.093,Z 401.772,A -85,B 0,C 180,E1 -8336.504,E2 -8336.504} C_VEL
LIN {X 0,Y 454.698,Z 409.12,A -85,B 0,C 180,E1 -8339.332,E2 -8339.332} C_VEL
LIN {X 0,Y 454.269,Z 418.596,A -85,B 0,C 180,E1 -8342.845,E2 -8342.845} C_VEL
LIN {X 0,Y 453.792,Z 427.982,A -85,B 0,C 180,E1 -8346.255,E2 -8346.255} C_VEL
LIN {X 0,Y 453.541,Z 436.034,A -85,B 0,C 180,E1 -8349.12,E2 -8349.12} C_VEL
LIN {X 0,Y 453.258,Z 444.097,A -85,B 0,C 180,E1 -8351.934,E2 -8351.934} C_VEL
LIN {X 0,Y 453.085,Z 450.344,A -85,B 0,C 180,E1 -8354.094,E2 -8354.094} C_VEL
LIN {X 0,Y 455.398,Z 464.28,A -85,B 0,C 180,E1 -8354.547,E2 -8354.547} C_VEL
LIN {X 0,Y 456.337,Z 471.998,A -85,B 0,C 180,E1 -8354.879,E2 -8354.879} C_VEL
LIN {X 0,Y 455.831,Z 484.364,A -85,B 0,C 180,E1 -8355.49,E2 -8355.49} C_VEL
LIN {X 0,Y 455.292,Z 496.261,A -85,B 0,C 180,E1 -8356.271,E2 -8356.271} C_VEL
LIN {X 0,Y 454.808,Z 506.812,A -85,B 0,C 180,E1 -8357.154,E2 -8357.154} C_VEL
LIN {X 0,Y 454.294,Z 516.691,A -85,B 0,C 180,E1 -8358.172,E2 -8358.172} C_VEL
LIN {X 0,Y 453.73,Z 525.581,A -85,B 0,C 180,E1 -8359.288,E2 -8359.288} C_VEL
LIN {X 0,Y 453.31,Z 534.265,A -85,B 0,C 180,E1 -8360.631,E2 -8360.631} C_VEL
LIN {X 0,Y 452.924,Z 541.206,A -85,B 0,C 180,E1 -8361.972,E2 -8361.972} C_VEL
LIN {X 0,Y 452.73,Z 547.349,A -85,B 0,C 180,E1 -8363.47,E2 -8363.47} C_VEL
LIN {X 0,Y 452.567,Z 552.384,A -85,B 0,C 180,E1 -8365.1,E2 -8365.1} C_VEL
LIN {X 0,Y 452.494,Z 555.341,A -85,B 0,C 180,E1 -8366.438,E2 -8366.438} C_VEL
LIN {X 0,Y 452.496,Z 556.751,A -85,B 0,C 180,E1 -8367.329,E2 -8367.329} C_VEL
LIN {X 0,Y 452.433,Z 558.367,A -85,B 0,C 180,E1 -8369.11,E2 -8369.11} C_VEL
LIN {X 0,Y 452.41,Z 558.584,A -85,B 0,C 180,E1 -8370,E2 -8370} C_VEL
LIN {X 0,Y 452.433,Z 558.367,A -85,B 0,C 180,E1 -8370.89,E2 -8370.89} C_VEL
LIN {X 0,Y 452.496,Z 556.754,A -85,B 0,C 180,E1 -8372.671,E2 -8372.671} C_VEL
LIN {X 0,Y 452.494,Z 555.345,A -85,B 0,C 180,E1 -8373.562,E2 -8373.562} C_VEL
LIN {X 0,Y 452.567,Z 552.386,A -85,B 0,C 180,E1 -8374.9,E2 -8374.9} C_VEL
LIN {X 0,Y 452.691,Z 547.508,A -85,B 0,C 180,E1 -8376.486,E2 -8376.486} C_VEL
LIN {X 0,Y 452.926,Z 541.208,A -85,B 0,C 180,E1 -8378.028,E2 -8378.028} C_VEL
LIN {X 0,Y 453.31,Z 534.266,A -85,B 0,C 180,E1 -8379.369,E2 -8379.369} C_VEL
LIN {X 0,Y 453.728,Z 525.583,A -85,B 0,C 180,E1 -8380.712,E2 -8380.712} C_VEL
LIN {X 0,Y 454.294,Z 516.693,A -85,B 0,C 180,E1 -8381.828,E2 -8381.828} C_VEL
LIN {X 0,Y 454.795,Z 506.803,A -85,B 0,C 180,E1 -8382.847,E2 -8382.847} C_VEL
LIN {X 0,Y 455.259,Z 496.265,A -85,B 0,C 180,E1 -8383.73,E2 -8383.73} C_VEL
LIN {X 0,Y 455.825,Z 484.364,A -85,B 0,C 180,E1 -8384.51,E2 -8384.51} C_VEL
LIN {X 0,Y 456.346,Z 471.993,A -85,B 0,C 180,E1 -8385.12,E2 -8385.12} C_VEL
LIN {X 0,Y 454.857,Z 460.96,A -85,B 0,C 180,E1 -8385.575,E2 -8385.575} C_VEL
LIN {X 0,Y 453.105,Z 450.067,A -85,B 0,C 180,E1 -8385.933,E2 -8385.933} C_VEL
LIN {X 0,Y 453.363,Z 441.373,A -85,B 0,C 180,E1 -8388.998,E2 -8388.998} C_VEL
LIN {X 0,Y 453.606,Z 433.297,A -85,B 0,C 180,E1 -8391.83,E2 -8391.83} C_VEL
LIN {X 0,Y 453.98,Z 423.931,A -85,B 0,C 180,E1 -8395.197,E2 -8395.197} C_VEL
LIN {X 0,Y 454.38,Z 415.798,A -85,B 0,C 180,E1 -8398.16,E2 -8398.16} C_VEL
LIN {X 0,Y 454.857,Z 406.098,A -85,B 0,C 180,E1 -8401.809,E2 -8401.809} C_VEL
LIN {X 0,Y 455.27,Z 398.377,A -85,B 0,C 180,E1 -8404.832,E2 -8404.832} C_VEL
LIN {X 0,Y 455.217,Z 394.079,A -85,B 0,C 180,E1 -8406.6,E2 -8406.6} C_VEL
LIN {X 0,Y 454.173,Z 387.825,A -85,B 0,C 180,E1 -8409.379,E2 -8409.379} C_VEL
LIN {X 0,Y 453.506,Z 383.997,A -85,B 0,C 180,E1 -8411.195,E2 -8411.195} C_VEL
LIN {X 0,Y 453.494,Z 384.003,A -85,B 0,C 180,E1 -8414.53,E2 -8414.53} C_VEL
LIN {X 0,Y 453.481,Z 383.994,A -85,B 0,C 180,E1 -8418.209,E2 -8418.209} C_VEL
LIN {X 0,Y 453.518,Z 383.996,A -85,B 0,C 180,E1 -8420.79,E2 -8420.79} C_VEL
LIN {X 0,Y 453.459,Z 384,A -85,B 0,C 180,E1 -8423.917,E2 -8423.917} C_VEL
LIN {X 0,Y 453.486,Z 383.999,A -85,B 0,C 180,E1 -8427.151,E2 -8427.151} C_VEL
LIN {X 0,Y 453.478,Z 383.996,A -85,B 0,C 180,E1 -8430.268,E2 -8430.268} C_VEL
LIN {X 0,Y 453.508,Z 383.993,A -85,B 0,C 180,E1 -8433.294,E2 -8433.294} C_VEL
LIN {X 0,Y 453.501,Z 383.997,A -85,B 0,C 180,E1 -8436.239,E2 -8436.239} C_VEL
LIN {X 0,Y 453.487,Z 383.998,A -85,B 0,C 180,E1 -8439.118,E2 -8439.118} C_VEL
LIN {X 0,Y 453.516,Z 383.992,A -85,B 0,C 180,E1 -8441.945,E2 -8441.945} C_VEL
LIN {X 0,Y 453.544,Z 383.991,A -85,B 0,C 180,E1 -8444.726,E2 -8444.726} C_VEL
LIN {X 0,Y 453.606,Z 383.981,A -85,B 0,C 180,E1 -8447.472,E2 -8447.472} C_VEL
LIN {X 0,Y 453.597,Z 383.984,A -85,B 0,C 180,E1 -8451.087,E2 -8451.087} C_VEL
LIN {X 0,Y 453.681,Z 383.972,A -85,B 0,C 180,E1 -8453.775,E2 -8453.775} C_VEL
LIN {X 0,Y 453.748,Z 383.961,A -85,B 0,C 180,E1 -8457.337,E2 -8457.337} C_VEL
LIN {X 0,Y 453.828,Z 383.956,A -85,B 0,C 180,E1 -8460,E2 -8460} C_VEL
LIN {X 0,Y 453.747,Z 383.965,A -85,B 0,C 180,E1 -8462.663,E2 -8462.663} C_VEL
LIN {X 0,Y 453.681,Z 383.973,A -85,B 0,C 180,E1 -8466.225,E2 -8466.225} C_VEL
LIN {X 0,Y 453.594,Z 383.981,A -85,B 0,C 180,E1 -8468.913,E2 -8468.913} C_VEL
LIN {X 0,Y 453.567,Z 383.986,A -85,B 0,C 180,E1 -8472.529,E2 -8472.529} C_VEL
LIN {X 0,Y 453.548,Z 383.99,A -85,B 0,C 180,E1 -8476.196,E2 -8476.196} C_VEL
LIN {X 0,Y 453.521,Z 383.991,A -85,B 0,C 180,E1 -8479.04,E2 -8479.04} C_VEL
LIN {X 0,Y 453.48,Z 383.998,A -85,B 0,C 180,E1 -8481.836,E2 -8481.836} C_VEL
LIN {X 0,Y 453.504,Z 383.993,A -85,B 0,C 180,E1 -8484.735,E2 -8484.735} C_VEL
LIN {X 0,Y 453.541,Z 383.991,A -85,B 0,C 180,E1 -8487.961,E2 -8487.961} C_VEL
LIN {X 0,Y 453.469,Z 383.999,A -85,B 0,C 180,E1 -8491.525,E2 -8491.525} C_VEL
LIN {X 0,Y 453.49,Z 383.994,A -85,B 0,C 180,E1 -8494.777,E2 -8494.777} C_VEL
LIN {X 0,Y 453.476,Z 383.997,A -85,B 0,C 180,E1 -8498.311,E2 -8498.311} C_VEL
LIN {X 0,Y 453.497,Z 383.995,A -85,B 0,C 180,E1 -8500.609,E2 -8500.609} C_VEL
LIN {X 0,Y 453.456,Z 384.002,A -85,B 0,C 180,E1 -8503.244,E2 -8503.244} C_VEL
LIN {X 0,Y 453.478,Z 384,A -85,B 0,C 180,E1 -8505.78,E2 -8505.78} C_VEL
LIN {X 0,Y 453.497,Z 383.994,A -85,B 0,C 180,E1 -8508.211,E2 -8508.211} C_VEL
LIN {X 0,Y 453.497,Z 383.993,A -85,B 0,C 180,E1 -8510.793,E2 -8510.793} C_VEL
LIN {X 0,Y 453.414,Z 384.006,A -85,B 0,C 180,E1 -8513.913,E2 -8513.913} C_VEL
LIN {X 0,Y 453.172,Z 384.04,A -85,B 0,C 180,E1 -8516.873,E2 -8516.873} C_VEL
LIN {X 0,Y 453.008,Z 384.085,A -85,B 0,C 180,E1 -8518.165,E2 -8518.165} C_VEL
LIN {X 0,Y 452.945,Z 387.084,A -85,B 0,C 180,E1 -8521.249,E2 -8521.249} C_VEL
LIN {X 0,Y 452.876,Z 389.946,A -85,B 0,C 180,E1 -8524.245,E2 -8524.245} C_VEL
LIN {X 0,Y 452.778,Z 392.837,A -85,B 0,C 180,E1 -8527.167,E2 -8527.167} C_VEL
LIN {X 0,Y 452.722,Z 395.837,A -85,B 0,C 180,E1 -8530.03,E2 -8530.03} C_VEL
LIN {X 0,Y 452.709,Z 398.975,A -85,B 0,C 180,E1 -8532.845,E2 -8532.845} C_VEL
LIN {X 0,Y 452.726,Z 400.56,A -85,B 0,C 180,E1 -8534.195,E2 -8534.195} C_VEL
LIN {X 0,Y 456.085,Z 414.563,A -85,B 0,C 180,E1 -8534.76,E2 -8534.76} C_VEL
LIN {X 0,Y 456.64,Z 418.567,A -85,B 0,C 180,E1 -8534.947,E2 -8534.947} C_VEL
LIN {X 0,Y 456.274,Z 429.79,A -85,B 0,C 180,E1 -8535.505,E2 -8535.505} C_VEL
LIN {X 0,Y 455.815,Z 441.368,A -85,B 0,C 180,E1 -8536.257,E2 -8536.257} C_VEL
LIN {X 0,Y 455.291,Z 452.424,A -85,B 0,C 180,E1 -8537.18,E2 -8537.18} C_VEL
LIN {X 0,Y 455.164,Z 454.344,A -85,B 0,C 180,E1 -8537.363,E2 -8537.363} C_VEL
LIN {X 0,Y 454.197,Z 458.998,A -85,B 0,C 180,E1 -8537.808,E2 -8537.808} C_VEL
LIN {X 0,Y 450.923,Z 466.289,A -85,B 0,C 180,E1 -8538.557,E2 -8538.557} C_VEL
LIN {X 0,Y 447.753,Z 473.031,A -85,B 0,C 180,E1 -8539.39,E2 -8539.39} C_VEL
LIN {X 0,Y 446.955,Z 476.8,A -85,B 0,C 180,E1 -8539.961,E2 -8539.961} C_VEL
LIN {X 0,Y 446.437,Z 484.658,A -85,B 0,C 180,E1 -8541.399,E2 -8541.399} C_VEL
LIN {X 0,Y 446.098,Z 490.574,A -85,B 0,C 180,E1 -8542.76,E2 -8542.76} C_VEL
LIN {X 0,Y 445.817,Z 495.251,A -85,B 0,C 180,E1 -8544.119,E2 -8544.119} C_VEL
LIN {X 0,Y 445.739,Z 498.823,A -85,B 0,C 180,E1 -8545.478,E2 -8545.478} C_VEL
LIN {X 0,Y 445.658,Z 500.671,A -85,B 0,C 180,E1 -8546.383,E2 -8546.383} C_VEL
LIN {X 0,Y 445.615,Z 502.063,A -85,B 0,C 180,E1 -8547.288,E2 -8547.288} C_VEL
LIN {X 0,Y 445.43,Z 503.67,A -85,B 0,C 180,E1 -8549.096,E2 -8549.096} C_VEL
LIN {X 0,Y 445.405,Z 503.904,A -85,B 0,C 180,E1 -8550,E2 -8550} C_VEL
LIN {X 0,Y 445.523,Z 503.133,A -85,B 0,C 180,E1 -8551.808,E2 -8551.808} C_VEL
LIN {X 0,Y 445.603,Z 502.172,A -85,B 0,C 180,E1 -8552.712,E2 -8552.712} C_VEL
LIN {X 0,Y 445.658,Z 500.827,A -85,B 0,C 180,E1 -8553.617,E2 -8553.617} C_VEL
LIN {X 0,Y 445.706,Z 497.988,A -85,B 0,C 180,E1 -8554.975,E2 -8554.975} C_VEL
LIN {X 0,Y 445.954,Z 494.126,A -85,B 0,C 180,E1 -8556.334,E2 -8556.334} C_VEL
LIN {X 0,Y 446.154,Z 489.15,A -85,B 0,C 180,E1 -8557.695,E2 -8557.695} C_VEL
LIN {X 0,Y 446.557,Z 482.875,A -85,B 0,C 180,E1 -8559.055,E2 -8559.055} C_VEL
LIN {X 0,Y 447.049,Z 475.015,A -85,B 0,C 180,E1 -8560.416,E2 -8560.416} C_VEL
LIN {X 0,Y 447.63,Z 465.233,A -85,B 0,C 180,E1 -8561.777,E2 -8561.777} C_VEL
LIN {X 0,Y 448.286,Z 454.956,A -85,B 0,C 180,E1 -8562.909,E2 -8562.909} C_VEL
LIN {X 0,Y 448.806,Z 443.506,A -85,B 0,C 180,E1 -8563.92,E2 -8563.92} C_VEL
LIN {X 0,Y 449.387,Z 431.807,A -85,B 0,C 180,E1 -8564.723,E2 -8564.723} C_VEL
LIN {X 0,Y 449.798,Z 419.783,A -85,B 0,C 180,E1 -8565.346,E2 -8565.346} C_VEL
LIN {X 0,Y 449.536,Z 416.944,A -85,B 0,C 180,E1 -8565.483,E2 -8565.483} C_VEL
LIN {X 0,Y 446.438,Z 404.188,A -85,B 0,C 180,E1 -8566.039,E2 -8566.039} C_VEL
LIN {X 0,Y 445.685,Z 400.893,A -85,B 0,C 180,E1 -8566.17,E2 -8566.17} C_VEL
LIN {X 0,Y 445.635,Z 397.354,A -85,B 0,C 180,E1 -8569.341,E2 -8569.341} C_VEL
LIN {X 0,Y 445.707,Z 394.288,A -85,B 0,C 180,E1 -8572.237,E2 -8572.237} C_VEL
LIN {X 0,Y 445.787,Z 391.327,A -85,B 0,C 180,E1 -8575.193,E2 -8575.193} C_VEL
LIN {X 0,Y 445.871,Z 388.358,A -85,B 0,C 180,E1 -8578.221,E2 -8578.221} C_VEL
LIN {X 0,Y 445.974,Z 385.428,A -85,B 0,C 180,E1 -8581.335,E2 -8581.335} C_VEL
LIN {X 0,Y 446.043,Z 384.926,A -85,B 0,C 180,E1 -8582.393,E2 -8582.393} C_VEL
LIN {X 0,Y 446.343,Z 384.885,A -85,B 0,C 180,E1 -8585.633,E2 -8585.633} C_VEL
LIN {X 0,Y 446.447,Z 384.873,A -85,B 0,C 180,E1 -8589.027,E2 -8589.027} C_VEL
LIN {X 0,Y 446.438,Z 384.877,A -85,B 0,C 180,E1 -8592.277,E2 -8592.277} C_VEL
LIN {X 0,Y 446.455,Z 384.872,A -85,B 0,C 180,E1 -8595.104,E2 -8595.104} C_VEL
LIN {X 0,Y 446.432,Z 384.878,A -85,B 0,C 180,E1 -8598.609,E2 -8598.609} C_VEL
LIN {X 0,Y 446.465,Z 384.87,A -85,B 0,C 180,E1 -8600.975,E2 -8600.975} C_VEL
LIN {X 0,Y 446.425,Z 384.878,A -85,B 0,C 180,E1 -8604.374,E2 -8604.374} C_VEL
LIN {X 0,Y 446.427,Z 384.876,A -85,B 0,C 180,E1 -8607.639,E2 -8607.639} C_VEL
LIN {X 0,Y 446.453,Z 384.873,A -85,B 0,C 180,E1 -8610.791,E2 -8610.791} C_VEL
LIN {X 0,Y 446.482,Z 384.87,A -85,B 0,C 180,E1 -8613.849,E2 -8613.849} C_VEL
LIN {X 0,Y 446.431,Z 384.873,A -85,B 0,C 180,E1 -8616.823,E2 -8616.823} C_VEL
LIN {X 0,Y 446.449,Z 384.876,A -85,B 0,C 180,E1 -8619.737,E2 -8619.737} C_VEL
LIN {X 0,Y 446.462,Z 384.872,A -85,B 0,C 180,E1 -8622.597,E2 -8622.597} C_VEL
LIN {X 0,Y 446.475,Z 384.871,A -85,B 0,C 180,E1 -8625.412,E2 -8625.412} C_VEL
LIN {X 0,Y 446.522,Z 384.865,A -85,B 0,C 180,E1 -8628.193,E2 -8628.193} C_VEL
LIN {X 0,Y 446.537,Z 384.86,A -85,B 0,C 180,E1 -8630.945,E2 -8630.945} C_VEL
LIN {X 0,Y 446.646,Z 384.851,A -85,B 0,C 180,E1 -8633.676,E2 -8633.676} C_VEL
LIN {X 0,Y 446.695,Z 384.844,A -85,B 0,C 180,E1 -8637.295,E2 -8637.295} C_VEL
LIN {X 0,Y 446.798,Z 384.832,A -85,B 0,C 180,E1 -8640,E2 -8640} C_VEL
LIN {X 0,Y 446.696,Z 384.839,A -85,B 0,C 180,E1 -8642.705,E2 -8642.705} C_VEL
LIN {X 0,Y 446.652,Z 384.847,A -85,B 0,C 180,E1 -8646.324,E2 -8646.324} C_VEL
LIN {X 0,Y 446.544,Z 384.863,A -85,B 0,C 180,E1 -8649.055,E2 -8649.055} C_VEL
LIN {X 0,Y 446.539,Z 384.861,A -85,B 0,C 180,E1 -8652.729,E2 -8652.729} C_VEL
LIN {X 0,Y 446.493,Z 384.865,A -85,B 0,C 180,E1 -8656.459,E2 -8656.459} C_VEL
LIN {X 0,Y 446.473,Z 384.873,A -85,B 0,C 180,E1 -8659.303,E2 -8659.303} C_VEL
LIN {X 0,Y 446.422,Z 384.876,A -85,B 0,C 180,E1 -8662.199,E2 -8662.199} C_VEL
LIN {X 0,Y 446.448,Z 384.874,A -85,B 0,C 180,E1 -8665.153,E2 -8665.153} C_VEL
LIN {X 0,Y 446.489,Z 384.865,A -85,B 0,C 180,E1 -8668.178,E2 -8668.178} C_VEL
LIN {X 0,Y 446.423,Z 384.876,A -85,B 0,C 180,E1 -8671.775,E2 -8671.775} C_VEL
LIN {X 0,Y 446.433,Z 384.876,A -85,B 0,C 180,E1 -8674.523,E2 -8674.523} C_VEL
LIN {X 0,Y 446.419,Z 384.876,A -85,B 0,C 180,E1 -8678.079,E2 -8678.079} C_VEL
LIN {X 0,Y 446.431,Z 384.877,A -85,B 0,C 180,E1 -8680.917,E2 -8680.917} C_VEL
LIN {X 0,Y 446.405,Z 384.88,A -85,B 0,C 180,E1 -8683.846,E2 -8683.846} C_VEL
LIN {X 0,Y 446.424,Z 384.879,A -85,B 0,C 180,E1 -8686.4,E2 -8686.4} C_VEL
LIN {X 0,Y 446.461,Z 384.955,A -85,B 0,C 180,E1 -8688.537,E2 -8688.537} C_VEL
LIN {X 0,Y 447.68,Z 391.709,A -85,B 0,C 180,E1 -8691.715,E2 -8691.715} C_VEL
LIN {X 0,Y 448.41,Z 396.891,A -85,B 0,C 180,E1 -8694.003,E2 -8694.003} C_VEL
LIN {X 0,Y 448.078,Z 403.531,A -85,B 0,C 180,E1 -8696.704,E2 -8696.704} C_VEL
LIN {X 0,Y 447.594,Z 411.292,A -85,B 0,C 180,E1 -8699.723,E2 -8699.723} C_VEL
LIN {X 0,Y 447.211,Z 419.692,A -85,B 0,C 180,E1 -8702.887,E2 -8702.887} C_VEL
LIN {X 0,Y 446.744,Z 429.081,A -85,B 0,C 180,E1 -8706.349,E2 -8706.349} C_VEL
LIN {X 0,Y 446.449,Z 437.108,A -85,B 0,C 180,E1 -8709.256,E2 -8709.256} C_VEL
LIN {X 0,Y 446.164,Z 445.052,A -85,B 0,C 180,E1 -8712.111,E2 -8712.111} C_VEL
LIN {X 0,Y 446.004,Z 450.075,A -85,B 0,C 180,E1 -8713.844,E2 -8713.844} C_VEL
LIN {X 0,Y 448.18,Z 463.003,A -85,B 0,C 180,E1 -8714.265,E2 -8714.265} C_VEL
LIN {X 0,Y 449.414,Z 472.869,A -85,B 0,C 180,E1 -8714.699,E2 -8714.699} C_VEL
LIN {X 0,Y 448.959,Z 483.932,A -85,B 0,C 180,E1 -8715.263,E2 -8715.263} C_VEL
LIN {X 0,Y 448.36,Z 495.827,A -85,B 0,C 180,E1 -8716.054,E2 -8716.054} C_VEL
LIN {X 0,Y 447.819,Z 506.805,A -85,B 0,C 180,E1 -8716.992,E2 -8716.992} C_VEL
LIN {X 0,Y 447.321,Z 516.257,A -85,B 0,C 180,E1 -8717.984,E2 -8717.984} C_VEL
LIN {X 0,Y 446.703,Z 525.146,A -85,B 0,C 180,E1 -8719.117,E2 -8719.117} C_VEL
LIN {X 0,Y 446.259,Z 533.83,A -85,B 0,C 180,E1 -8720.482,E2 -8720.482} C_VEL
LIN {X 0,Y 445.884,Z 540.773,A -85,B 0,C 180,E1 -8721.845,E2 -8721.845} C_VEL
LIN {X 0,Y 445.65,Z 546.345,A -85,B 0,C 180,E1 -8723.208,E2 -8723.208} C_VEL
LIN {X 0,Y 445.541,Z 550.717,A -85,B 0,C 180,E1 -8724.569,E2 -8724.569} C_VEL
LIN {X 0,Y 445.427,Z 553.029,A -85,B 0,C 180,E1 -8725.475,E2 -8725.475} C_VEL
LIN {X 0,Y 445.398,Z 554.908,A -85,B 0,C 180,E1 -8726.381,E2 -8726.381} C_VEL
LIN {X 0,Y 445.423,Z 556.32,A -85,B 0,C 180,E1 -8727.287,E2 -8727.287} C_VEL
LIN {X 0,Y 445.372,Z 557.937,A -85,B 0,C 180,E1 -8729.096,E2 -8729.096} C_VEL
LIN {X 0,Y 445.349,Z 558.154,A -85,B 0,C 180,E1 -8730,E2 -8730} C_VEL
LIN {X 0,Y 445.372,Z 557.938,A -85,B 0,C 180,E1 -8730.904,E2 -8730.904} C_VEL
LIN {X 0,Y 445.423,Z 556.323,A -85,B 0,C 180,E1 -8732.713,E2 -8732.713} C_VEL
LIN {X 0,Y 445.398,Z 554.912,A -85,B 0,C 180,E1 -8733.619,E2 -8733.619} C_VEL
LIN {X 0,Y 445.5,Z 551.954,A -85,B 0,C 180,E1 -8734.977,E2 -8734.977} C_VEL
LIN {X 0,Y 445.587,Z 547.57,A -85,B 0,C 180,E1 -8736.451,E2 -8736.451} C_VEL
LIN {X 0,Y 445.804,Z 541.792,A -85,B 0,C 180,E1 -8737.929,E2 -8737.929} C_VEL
LIN {X 0,Y 446.186,Z 535.075,A -85,B 0,C 180,E1 -8739.291,E2 -8739.291} C_VEL
LIN {X 0,Y 446.628,Z 526.744,A -85,B 0,C 180,E1 -8740.655,E2 -8740.655} C_VEL
LIN {X 0,Y 447.187,Z 518.217,A -85,B 0,C 180,E1 -8741.789,E2 -8741.789} C_VEL
LIN {X 0,Y 447.72,Z 508.415,A -85,B 0,C 180,E1 -8742.854,E2 -8742.854} C_VEL
LIN {X 0,Y 448.263,Z 497.265,A -85,B 0,C 180,E1 -8743.833,E2 -8743.833} C_VEL
LIN {X 0,Y 448.831,Z 485.858,A -85,B 0,C 180,E1 -8744.625,E2 -8744.625} C_VEL
LIN {X 0,Y 449.385,Z 474.169,A -85,B 0,C 180,E1 -8745.244,E2 -8745.244} C_VEL
LIN {X 0,Y 449.224,Z 470.236,A -85,B 0,C 180,E1 -8745.424,E2 -8745.424} C_VEL
LIN {X 0,Y 447.139,Z 457.136,A -85,B 0,C 180,E1 -8745.95,E2 -8745.95} C_VEL
LIN {X 0,Y 446.007,Z 449.717,A -85,B 0,C 180,E1 -8746.182,E2 -8746.182} C_VEL
LIN {X 0,Y 446.327,Z 441.037,A -85,B 0,C 180,E1 -8749.31,E2 -8749.31} C_VEL
LIN {X 0,Y 446.642,Z 431.74,A -85,B 0,C 180,E1 -8752.676,E2 -8752.676} C_VEL
LIN {X 0,Y 447.083,Z 422.341,A -85,B 0,C 180,E1 -8756.114,E2 -8756.114} C_VEL
LIN {X 0,Y 447.422,Z 414.235,A -85,B 0,C 180,E1 -8759.14,E2 -8759.14} C_VEL
LIN {X 0,Y 447.917,Z 406.179,A -85,B 0,C 180,E1 -8762.241,E2 -8762.241} C_VEL
LIN {X 0,Y 448.37,Z 398.286,A -85,B 0,C 180,E1 -8765.405,E2 -8765.405} C_VEL
LIN {X 0,Y 448.187,Z 394.788,A -85,B 0,C 180,E1 -8766.895,E2 -8766.895} C_VEL
LIN {X 0,Y 446.986,Z 387.676,A -85,B 0,C 180,E1 -8770.139,E2 -8770.139} C_VEL
LIN {X 0,Y 446.456,Z 384.877,A -85,B 0,C 180,E1 -8771.539,E2 -8771.539} C_VEL
LIN {X 0,Y 446.457,Z 384.881,A -85,B 0,C 180,E1 -8775.103,E2 -8775.103} C_VEL
LIN {X 0,Y 446.43,Z 384.876,A -85,B 0,C 180,E1 -8778.609,E2 -8778.609} C_VEL
LIN {X 0,Y 446.464,Z 384.873,A -85,B 0,C 180,E1 -8780.975,E2 -8780.975} C_VEL
LIN {X 0,Y 446.424,Z 384.878,A -85,B 0,C 180,E1 -8784.374,E2 -8784.374} C_VEL
LIN {X 0,Y 446.425,Z 384.875,A -85,B 0,C 180,E1 -8787.639,E2 -8787.639} C_VEL
LIN {X 0,Y 446.452,Z 384.876,A -85,B 0,C 180,E1 -8790.791,E2 -8790.791} C_VEL
LIN {X 0,Y 446.481,Z 384.868,A -85,B 0,C 180,E1 -8793.849,E2 -8793.849} C_VEL
LIN {X 0,Y 446.429,Z 384.877,A -85,B 0,C 180,E1 -8796.823,E2 -8796.823} C_VEL
LIN {X 0,Y 446.448,Z 384.872,A -85,B 0,C 180,E1 -8799.737,E2 -8799.737} C_VEL
LIN {X 0,Y 446.468,Z 384.873,A -85,B 0,C 180,E1 -8802.597,E2 -8802.597} C_VEL
LIN {X 0,Y 446.474,Z 384.868,A -85,B 0,C 180,E1 -8805.413,E2 -8805.413} C_VEL
LIN {X 0,Y 446.543,Z 384.864,A -85,B 0,C 180,E1 -8808.194,E2 -8808.194} C_VEL
LIN {X 0,Y 446.604,Z 384.854,A -85,B 0,C 180,E1 -8811.858,E2 -8811.858} C_VEL
LIN {X 0,Y 446.649,Z 384.852,A -85,B 0,C 180,E1 -8814.583,E2 -8814.583} C_VEL
LIN {X 0,Y 446.668,Z 384.848,A -85,B 0,C 180,E1 -8818.197,E2 -8818.197} C_VEL
LIN {X 0,Y 446.798,Z 384.831,A -85,B 0,C 180,E1 -8820,E2 -8820} C_VEL
LIN {X 0,Y 446.694,Z 384.844,A -85,B 0,C 180,E1 -8822.705,E2 -8822.705} C_VEL
LIN {X 0,Y 446.651,Z 384.85,A -85,B 0,C 180,E1 -8826.324,E2 -8826.324} C_VEL
LIN {X 0,Y 446.54,Z 384.859,A -85,B 0,C 180,E1 -8829.055,E2 -8829.055} C_VEL
LIN {X 0,Y 446.525,Z 384.863,A -85,B 0,C 180,E1 -8832.73,E2 -8832.73} C_VEL
LIN {X 0,Y 446.499,Z 384.868,A -85,B 0,C 180,E1 -8836.228,E2 -8836.228} C_VEL
LIN {X 0,Y 446.472,Z 384.87,A -85,B 0,C 180,E1 -8839.303,E2 -8839.303} C_VEL
LIN {X 0,Y 446.422,Z 384.879,A -85,B 0,C 180,E1 -8842.2,E2 -8842.2} C_VEL
LIN {X 0,Y 446.447,Z 384.872,A -85,B 0,C 180,E1 -8845.153,E2 -8845.153} C_VEL
LIN {X 0,Y 446.488,Z 384.869,A -85,B 0,C 180,E1 -8848.179,E2 -8848.179} C_VEL
LIN {X 0,Y 446.422,Z 384.877,A -85,B 0,C 180,E1 -8851.775,E2 -8851.775} C_VEL
LIN {X 0,Y 446.432,Z 384.874,A -85,B 0,C 180,E1 -8854.523,E2 -8854.523} C_VEL
LIN {X 0,Y 446.433,Z 384.875,A -85,B 0,C 180,E1 -8858.082,E2 -8858.082} C_VEL
LIN {X 0,Y 446.43,Z 384.875,A -85,B 0,C 180,E1 -8860.918,E2 -8860.918} C_VEL
LIN {X 0,Y 446.401,Z 384.881,A -85,B 0,C 180,E1 -8863.846,E2 -8863.846} C_VEL
LIN {X 0,Y 446.449,Z 384.872,A -85,B 0,C 180,E1 -8866.397,E2 -8866.397} C_VEL
LIN {X 0,Y 446.446,Z 384.875,A -85,B 0,C 180,E1 -8869.802,E2 -8869.802} C_VEL
LIN {X 0,Y 446.409,Z 384.878,A -85,B 0,C 180,E1 -8872.121,E2 -8872.121} C_VEL
LIN {X 0,Y 446.319,Z 384.89,A -85,B 0,C 180,E1 -8874.967,E2 -8874.967} C_VEL
LIN {X 0,Y 445.959,Z 385.012,A -85,B 0,C 180,E1 -8878.321,E2 -8878.321} C_VEL
LIN {X 0,Y 445.871,Z 388.319,A -85,B 0,C 180,E1 -8881.779,E2 -8881.779} C_VEL
LIN {X 0,Y 445.795,Z 391.245,A -85,B 0,C 180,E1 -8884.808,E2 -8884.808} C_VEL
LIN {X 0,Y 445.71,Z 394.18,A -85,B 0,C 180,E1 -8887.763,E2 -8887.763} C_VEL
LIN {X 0,Y 445.704,Z 397.715,A -85,B 0,C 180,E1 -8891.103,E2 -8891.103} C_VEL
LIN {X 0,Y 445.688,Z 400.97,A -85,B 0,C 180,E1 -8893.942,E2 -8893.942} C_VEL
LIN {X 0,Y 448.916,Z 414.338,A -85,B 0,C 180,E1 -8894.484,E2 -8894.484} C_VEL
LIN {X 0,Y 449.817,Z 419.008,A -85,B 0,C 180,E1 -8894.713,E2 -8894.713} C_VEL
LIN {X 0,Y 449.44,Z 430.229,A -85,B 0,C 180,E1 -8895.279,E2 -8895.279} C_VEL
LIN {X 0,Y 448.94,Z 442.179,A -85,B 0,C 180,E1 -8896.071,E2 -8896.071} C_VEL
LIN {X 0,Y 448.402,Z 452.86,A -85,B 0,C 180,E1 -8896.979,E2 -8896.979} C_VEL
LIN {X 0,Y 447.864,Z 462.547,A -85,B 0,C 180,E1 -8897.999,E2 -8897.999} C_VEL
LIN {X 0,Y 447.265,Z 471.359,A -85,B 0,C 180,E1 -8899.131,E2 -8899.131} C_VEL
LIN {X 0,Y 446.955,Z 476.8,A -85,B 0,C 180,E1 -8899.961,E2 -8899.961} C_VEL
LIN {X 0,Y 446.144,Z 480.39,A -85,B 0,C 180,E1 -8900.555,E2 -8900.555} C_VEL
LIN {X 0,Y 442.942,Z 485.87,A -85,B 0,C 180,E1 -8901.539,E2 -8901.539} C_VEL
LIN {X 0,Y 439.749,Z 490.719,A -85,B 0,C 180,E1 -8902.586,E2 -8902.586} C_VEL
LIN {X 0,Y 438.965,Z 493.267,A -85,B 0,C 180,E1 -8903.272,E2 -8903.272} C_VEL
LIN {X 0,Y 438.629,Z 498.207,A -85,B 0,C 180,E1 -8904.944,E2 -8904.944} C_VEL
LIN {X 0,Y 438.599,Z 501.103,A -85,B 0,C 180,E1 -8906.325,E2 -8906.325} C_VEL
LIN {X 0,Y 438.537,Z 502.495,A -85,B 0,C 180,E1 -8907.244,E2 -8907.244} C_VEL
LIN {X 0,Y 438.37,Z 504.1,A -85,B 0,C 180,E1 -8909.081,E2 -8909.081} C_VEL
LIN {X 0,Y 438.343,Z 504.334,A -85,B 0,C 180,E1 -8910,E2 -8910} C_VEL
LIN {X 0,Y 438.468,Z 503.563,A -85,B 0,C 180,E1 -8911.837,E2 -8911.837} C_VEL
LIN {X 0,Y 438.599,Z 501.257,A -85,B 0,C 180,E1 -8913.675,E2 -8913.675} C_VEL
LIN {X 0,Y 438.627,Z 498.42,A -85,B 0,C 180,E1 -8915.056,E2 -8915.056} C_VEL
LIN {X 0,Y 438.914,Z 494.556,A -85,B 0,C 180,E1 -8916.436,E2 -8916.436} C_VEL
LIN {X 0,Y 439.125,Z 489.58,A -85,B 0,C 180,E1 -8917.819,E2 -8917.819} C_VEL
LIN {X 0,Y 439.567,Z 483.303,A -85,B 0,C 180,E1 -8919.2,E2 -8919.2} C_VEL
LIN {X 0,Y 440.084,Z 475.443,A -85,B 0,C 180,E1 -8920.583,E2 -8920.583} C_VEL
LIN {X 0,Y 440.694,Z 465.661,A -85,B 0,C 180,E1 -8921.965,E2 -8921.965} C_VEL
LIN {X 0,Y 441.402,Z 455.389,A -85,B 0,C 180,E1 -8923.113,E2 -8923.113} C_VEL
LIN {X 0,Y 441.942,Z 443.967,A -85,B 0,C 180,E1 -8924.138,E2 -8924.138} C_VEL
LIN {X 0,Y 442.543,Z 432.23,A -85,B 0,C 180,E1 -8924.955,E2 -8924.955} C_VEL
LIN {X 0,Y 442.988,Z 420.203,A -85,B 0,C 180,E1 -8925.588,E2 -8925.588} C_VEL
LIN {X 0,Y 440.53,Z 408.8,A -85,B 0,C 180,E1 -8926.132,E2 -8926.132} C_VEL
LIN {X 0,Y 438.601,Z 401.312,A -85,B 0,C 180,E1 -8926.436,E2 -8926.436} C_VEL
LIN {X 0,Y 438.588,Z 397.736,A -85,B 0,C 180,E1 -8929.664,E2 -8929.664} C_VEL
LIN {X 0,Y 438.647,Z 394.641,A -85,B 0,C 180,E1 -8932.615,E2 -8932.615} C_VEL
LIN {X 0,Y 438.725,Z 391.654,A -85,B 0,C 180,E1 -8935.628,E2 -8935.628} C_VEL
LIN {X 0,Y 438.803,Z 388.657,A -85,B 0,C 180,E1 -8938.718,E2 -8938.718} C_VEL
LIN {X 0,Y 438.95,Z 385.809,A -85,B 0,C 180,E1 -8941.942,E2 -8941.942} C_VEL
LIN {X 0,Y 439.305,Z 385.762,A -85,B 0,C 180,E1 -8945.323,E2 -8945.323} C_VEL
LIN {X 0,Y 439.381,Z 385.757,A -85,B 0,C 180,E1 -8948.596,E2 -8948.596} C_VEL
LIN {X 0,Y 439.392,Z 385.75,A -85,B 0,C 180,E1 -8951.257,E2 -8951.257} C_VEL
LIN {X 0,Y 439.403,Z 385.751,A -85,B 0,C 180,E1 -8954.73,E2 -8954.73} C_VEL
LIN {X 0,Y 439.399,Z 385.752,A -85,B 0,C 180,E1 -8957.796,E2 -8957.796} C_VEL
LIN {X 0,Y 439.441,Z 385.747,A -85,B 0,C 180,E1 -8960.229,E2 -8960.229} C_VEL
LIN {X 0,Y 439.381,Z 385.752,A -85,B 0,C 180,E1 -8963.713,E2 -8963.713} C_VEL
LIN {X 0,Y 439.376,Z 385.753,A -85,B 0,C 180,E1 -8967.054,E2 -8967.054} C_VEL
LIN {X 0,Y 439.387,Z 385.754,A -85,B 0,C 180,E1 -8970.274,E2 -8970.274} C_VEL
LIN {X 0,Y 439.432,Z 385.747,A -85,B 0,C 180,E1 -8973.396,E2 -8973.396} C_VEL
LIN {X 0,Y 439.389,Z 385.752,A -85,B 0,C 180,E1 -8976.43,E2 -8976.43} C_VEL
LIN {X 0,Y 439.393,Z 385.751,A -85,B 0,C 180,E1 -8979.397,E2 -8979.397} C_VEL
LIN {X 0,Y 439.431,Z 385.749,A -85,B 0,C 180,E1 -8982.309,E2 -8982.309} C_VEL
LIN {X 0,Y 439.453,Z 385.744,A -85,B 0,C 180,E1 -8985.174,E2 -8985.174} C_VEL
LIN {X 0,Y 439.488,Z 385.744,A -85,B 0,C 180,E1 -8988.001,E2 -8988.001} C_VEL
LIN {X 0,Y 439.509,Z 385.741,A -85,B 0,C 180,E1 -8991.725,E2 -8991.725} C_VEL
LIN {X 0,Y 439.624,Z 385.723,A -85,B 0,C 180,E1 -8994.496,E2 -8994.496} C_VEL
LIN {X 0,Y 439.639,Z 385.723,A -85,B 0,C 180,E1 -8998.168,E2 -8998.168} C_VEL
LIN {X 0,Y 439.767,Z 385.707,A -85,B 0,C 180,E1 -9000,E2 -9000} C_VEL
LIN {X 0,Y 439.645,Z 385.718,A -85,B 0,C 180,E1 -9002.749,E2 -9002.749} C_VEL
LIN {X 0,Y 439.623,Z 385.722,A -85,B 0,C 180,E1 -9006.425,E2 -9006.425} C_VEL
LIN {X 0,Y 439.506,Z 385.74,A -85,B 0,C 180,E1 -9009.201,E2 -9009.201} C_VEL
LIN {X 0,Y 439.509,Z 385.737,A -85,B 0,C 180,E1 -9012.726,E2 -9012.726} C_VEL
LIN {X 0,Y 439.451,Z 385.742,A -85,B 0,C 180,E1 -9016.348,E2 -9016.348} C_VEL
LIN {X 0,Y 439.407,Z 385.751,A -85,B 0,C 180,E1 -9019.626,E2 -9019.626} C_VEL
LIN {X 0,Y 439.368,Z 385.755,A -85,B 0,C 180,E1 -9022.575,E2 -9022.575} C_VEL
LIN {X 0,Y 439.402,Z 385.753,A -85,B 0,C 180,E1 -9025.585,E2 -9025.585} C_VEL
LIN {X 0,Y 439.422,Z 385.747,A -85,B 0,C 180,E1 -9028.673,E2 -9028.673} C_VEL
LIN {X 0,Y 439.374,Z 385.753,A -85,B 0,C 180,E1 -9032.03,E2 -9032.03} C_VEL
LIN {X 0,Y 439.398,Z 385.753,A -85,B 0,C 180,E1 -9035.34,E2 -9035.34} C_VEL
LIN {X 0,Y 439.387,Z 385.753,A -85,B 0,C 180,E1 -9038.595,E2 -9038.595} C_VEL
LIN {X 0,Y 439.392,Z 385.756,A -85,B 0,C 180,E1 -9041.257,E2 -9041.257} C_VEL
LIN {X 0,Y 439.406,Z 385.754,A -85,B 0,C 180,E1 -9044.729,E2 -9044.729} C_VEL
LIN {X 0,Y 439.424,Z 385.768,A -85,B 0,C 180,E1 -9048.172,E2 -9048.172} C_VEL
LIN {X 0,Y 440.62,Z 392.481,A -85,B 0,C 180,E1 -9051.404,E2 -9051.404} C_VEL
LIN {X 0,Y 441.445,Z 398.025,A -85,B 0,C 180,E1 -9053.909,E2 -9053.909} C_VEL
LIN {X 0,Y 441.092,Z 404.649,A -85,B 0,C 180,E1 -9056.654,E2 -9056.654} C_VEL
LIN {X 0,Y 440.617,Z 411.747,A -85,B 0,C 180,E1 -9059.465,E2 -9059.465} C_VEL
LIN {X 0,Y 440.242,Z 419.43,A -85,B 0,C 180,E1 -9062.422,E2 -9062.422} C_VEL
LIN {X 0,Y 439.814,Z 427.937,A -85,B 0,C 180,E1 -9065.621,E2 -9065.621} C_VEL
LIN {X 0,Y 439.419,Z 436.801,A -85,B 0,C 180,E1 -9068.908,E2 -9068.908} C_VEL
LIN {X 0,Y 439.12,Z 444.706,A -85,B 0,C 180,E1 -9071.814,E2 -9071.814} C_VEL
LIN {X 0,Y 438.972,Z 449.747,A -85,B 0,C 180,E1 -9073.58,E2 -9073.58} C_VEL
LIN {X 0,Y 441.122,Z 462.931,A -85,B 0,C 180,E1 -9074.019,E2 -9074.019} C_VEL
LIN {X 0,Y 442.533,Z 472.434,A -85,B 0,C 180,E1 -9074.455,E2 -9074.455} C_VEL
LIN {X 0,Y 442.095,Z 483.499,A -85,B 0,C 180,E1 -9075.029,E2 -9075.029} C_VEL
LIN {X 0,Y 441.438,Z 495.392,A -85,B 0,C 180,E1 -9075.831,E2 -9075.831} C_VEL
LIN {X 0,Y 440.82,Z 506.846,A -85,B 0,C 180,E1 -9076.829,E2 -9076.829} C_VEL
LIN {X 0,Y 440.217,Z 517.781,A -85,B 0,C 180,E1 -9078.021,E2 -9078.021} C_VEL
LIN {X 0,Y 439.612,Z 526.308,A -85,B 0,C 180,E1 -9079.173,E2 -9079.173} C_VEL
LIN {X 0,Y 439.152,Z 534.64,A -85,B 0,C 180,E1 -9080.559,E2 -9080.559} C_VEL
LIN {X 0,Y 438.752,Z 541.357,A -85,B 0,C 180,E1 -9081.943,E2 -9081.943} C_VEL
LIN {X 0,Y 438.546,Z 547.517,A -85,B 0,C 180,E1 -9083.559,E2 -9083.559} C_VEL
LIN {X 0,Y 438.434,Z 551.521,A -85,B 0,C 180,E1 -9084.942,E2 -9084.942} C_VEL
LIN {X 0,Y 438.303,Z 554.475,A -85,B 0,C 180,E1 -9086.323,E2 -9086.323} C_VEL
LIN {X 0,Y 438.351,Z 555.888,A -85,B 0,C 180,E1 -9087.243,E2 -9087.243} C_VEL
LIN {X 0,Y 438.283,Z 557.505,A -85,B 0,C 180,E1 -9089.081,E2 -9089.081} C_VEL
LIN {X 0,Y 438.29,Z 557.724,A -85,B 0,C 180,E1 -9090,E2 -9090} C_VEL
LIN {X 0,Y 438.283,Z 557.506,A -85,B 0,C 180,E1 -9090.919,E2 -9090.919} C_VEL
LIN {X 0,Y 438.351,Z 555.892,A -85,B 0,C 180,E1 -9092.757,E2 -9092.757} C_VEL
LIN {X 0,Y 438.303,Z 554.479,A -85,B 0,C 180,E1 -9093.677,E2 -9093.677} C_VEL
LIN {X 0,Y 438.434,Z 551.522,A -85,B 0,C 180,E1 -9095.058,E2 -9095.058} C_VEL
LIN {X 0,Y 438.506,Z 547.513,A -85,B 0,C 180,E1 -9096.442,E2 -9096.442} C_VEL
LIN {X 0,Y 438.753,Z 541.358,A -85,B 0,C 180,E1 -9098.057,E2 -9098.057} C_VEL
LIN {X 0,Y 439.152,Z 534.641,A -85,B 0,C 180,E1 -9099.441,E2 -9099.441} C_VEL
LIN {X 0,Y 439.611,Z 526.309,A -85,B 0,C 180,E1 -9100.827,E2 -9100.827} C_VEL
LIN {X 0,Y 440.212,Z 517.783,A -85,B 0,C 180,E1 -9101.979,E2 -9101.979} C_VEL
LIN {X 0,Y 440.745,Z 508.224,A -85,B 0,C 180,E1 -9103.037,E2 -9103.037} C_VEL
LIN {X 0,Y 441.332,Z 496.83,A -85,B 0,C 180,E1 -9104.055,E2 -9104.055} C_VEL
LIN {X 0,Y 441.956,Z 485.425,A -85,B 0,C 180,E1 -9104.858,E2 -9104.858} C_VEL
LIN {X 0,Y 442.508,Z 473.734,A -85,B 0,C 180,E1 -9105.487,E2 -9105.487} C_VEL
LIN {X 0,Y 441.052,Z 462.542,A -85,B 0,C 180,E1 -9105.996,E2 -9105.996} C_VEL
LIN {X 0,Y 438.957,Z 449.365,A -85,B 0,C 180,E1 -9106.452,E2 -9106.452} C_VEL
LIN {X 0,Y 439.258,Z 440.727,A -85,B 0,C 180,E1 -9109.633,E2 -9109.633} C_VEL
LIN {X 0,Y 439.636,Z 431.494,A -85,B 0,C 180,E1 -9113.058,E2 -9113.058} C_VEL
LIN {X 0,Y 440.085,Z 422.067,A -85,B 0,C 180,E1 -9116.561,E2 -9116.561} C_VEL
LIN {X 0,Y 440.387,Z 415.323,A -85,B 0,C 180,E1 -9119.126,E2 -9119.126} C_VEL
LIN {X 0,Y 440.919,Z 407.099,A -85,B 0,C 180,E1 -9122.35,E2 -9122.35} C_VEL
LIN {X 0,Y 441.331,Z 400.647,A -85,B 0,C 180,E1 -9124.98,E2 -9124.98} C_VEL
LIN {X 0,Y 441.284,Z 396.748,A -85,B 0,C 180,E1 -9126.641,E2 -9126.641} C_VEL
LIN {X 0,Y 440.405,Z 391.403,A -85,B 0,C 180,E1 -9129.088,E2 -9129.088} C_VEL
LIN {X 0,Y 439.404,Z 385.756,A -85,B 0,C 180,E1 -9131.829,E2 -9131.829} C_VEL
LIN {X 0,Y 439.405,Z 385.759,A -85,B 0,C 180,E1 -9135.271,E2 -9135.271} C_VEL
LIN {X 0,Y 439.391,Z 385.754,A -85,B 0,C 180,E1 -9138.743,E2 -9138.743} C_VEL
LIN {X 0,Y 439.388,Z 385.752,A -85,B 0,C 180,E1 -9141.606,E2 -9141.606} C_VEL
LIN {X 0,Y 439.403,Z 385.752,A -85,B 0,C 180,E1 -9144.844,E2 -9144.844} C_VEL
LIN {X 0,Y 439.376,Z 385.754,A -85,B 0,C 180,E1 -9148.14,E2 -9148.14} C_VEL
LIN {X 0,Y 439.435,Z 385.744,A -85,B 0,C 180,E1 -9151.598,E2 -9151.598} C_VEL
LIN {X 0,Y 439.401,Z 385.753,A -85,B 0,C 180,E1 -9154.415,E2 -9154.415} C_VEL
LIN {X 0,Y 439.367,Z 385.755,A -85,B 0,C 180,E1 -9157.425,E2 -9157.425} C_VEL
LIN {X 0,Y 439.445,Z 385.748,A -85,B 0,C 180,E1 -9160.663,E2 -9160.663} C_VEL
LIN {X 0,Y 439.466,Z 385.743,A -85,B 0,C 180,E1 -9164.225,E2 -9164.225} C_VEL
LIN {X 0,Y 439.511,Z 385.738,A -85,B 0,C 180,E1 -9168.002,E2 -9168.002} C_VEL
LIN {X 0,Y 439.552,Z 385.732,A -85,B 0,C 180,E1 -9171.726,E2 -9171.726} C_VEL
LIN {X 0,Y 439.624,Z 385.726,A -85,B 0,C 180,E1 -9174.496,E2 -9174.496} C_VEL
LIN {X 0,Y 439.638,Z 385.723,A -85,B 0,C 180,E1 -9178.168,E2 -9178.168} C_VEL
LIN {X 0,Y 439.768,Z 385.707,A -85,B 0,C 180,E1 -9180,E2 -9180} C_VEL
LIN {X 0,Y 439.643,Z 385.723,A -85,B 0,C 180,E1 -9182.749,E2 -9182.749} C_VEL
LIN {X 0,Y 439.622,Z 385.726,A -85,B 0,C 180,E1 -9186.425,E2 -9186.425} C_VEL
LIN {X 0,Y 439.502,Z 385.736,A -85,B 0,C 180,E1 -9189.202,E2 -9189.202} C_VEL
LIN {X 0,Y 439.469,Z 385.741,A -85,B 0,C 180,E1 -9192.938,E2 -9192.938} C_VEL
LIN {X 0,Y 439.45,Z 385.746,A -85,B 0,C 180,E1 -9196.348,E2 -9196.348} C_VEL
LIN {X 0,Y 439.406,Z 385.751,A -85,B 0,C 180,E1 -9199.626,E2 -9199.626} C_VEL
LIN {X 0,Y 439.368,Z 385.754,A -85,B 0,C 180,E1 -9202.575,E2 -9202.575} C_VEL
LIN {X 0,Y 439.401,Z 385.752,A -85,B 0,C 180,E1 -9205.585,E2 -9205.585} C_VEL
LIN {X 0,Y 439.421,Z 385.748,A -85,B 0,C 180,E1 -9208.673,E2 -9208.673} C_VEL
LIN {X 0,Y 439.374,Z 385.757,A -85,B 0,C 180,E1 -9212.031,E2 -9212.031} C_VEL
LIN {X 0,Y 439.397,Z 385.751,A -85,B 0,C 180,E1 -9215.34,E2 -9215.34} C_VEL
LIN {X 0,Y 439.393,Z 385.751,A -85,B 0,C 180,E1 -9218.594,E2 -9218.594} C_VEL
LIN {X 0,Y 439.391,Z 385.753,A -85,B 0,C 180,E1 -9221.257,E2 -9221.257} C_VEL
LIN {X 0,Y 439.403,Z 385.75,A -85,B 0,C 180,E1 -9224.729,E2 -9224.729} C_VEL
LIN {X 0,Y 439.414,Z 385.752,A -85,B 0,C 180,E1 -9227.798,E2 -9227.798} C_VEL
LIN {X 0,Y 439.428,Z 385.746,A -85,B 0,C 180,E1 -9230.227,E2 -9230.227} C_VEL
LIN {X 0,Y 439.319,Z 385.762,A -85,B 0,C 180,E1 -9233.707,E2 -9233.707} C_VEL
LIN {X 0,Y 439.12,Z 385.789,A -85,B 0,C 180,E1 -9236.331,E2 -9236.331} C_VEL
LIN {X 0,Y 438.938,Z 385.812,A -85,B 0,C 180,E1 -9238.104,E2 -9238.104} C_VEL
LIN {X 0,Y 438.801,Z 388.584,A -85,B 0,C 180,E1 -9241.282,E2 -9241.282} C_VEL
LIN {X 0,Y 438.741,Z 391.591,A -85,B 0,C 180,E1 -9244.374,E2 -9244.374} C_VEL
LIN {X 0,Y 438.649,Z 394.534,A -85,B 0,C 180,E1 -9247.386,E2 -9247.386} C_VEL
LIN {X 0,Y 438.659,Z 398.282,A -85,B 0,C 180,E1 -9250.957,E2 -9250.957} C_VEL
LIN {X 0,Y 438.629,Z 401.535,A -85,B 0,C 180,E1 -9253.679,E2 -9253.679} C_VEL
LIN {X 0,Y 441.917,Z 414.717,A -85,B 0,C 180,E1 -9254.229,E2 -9254.229} C_VEL
LIN {X 0,Y 442.948,Z 419.453,A -85,B 0,C 180,E1 -9254.47,E2 -9254.47} C_VEL
LIN {X 0,Y 442.607,Z 430.667,A -85,B 0,C 180,E1 -9255.047,E2 -9255.047} C_VEL
LIN {X 0,Y 442.092,Z 442.017,A -85,B 0,C 180,E1 -9255.805,E2 -9255.805} C_VEL
LIN {X 0,Y 441.519,Z 453.295,A -85,B 0,C 180,E1 -9256.773,E2 -9256.773} C_VEL
LIN {X 0,Y 440.934,Z 462.983,A -85,B 0,C 180,E1 -9257.808,E2 -9257.808} C_VEL
LIN {X 0,Y 440.325,Z 471.793,A -85,B 0,C 180,E1 -9258.958,E2 -9258.958} C_VEL
LIN {X 0,Y 439.804,Z 480.378,A -85,B 0,C 180,E1 -9260.341,E2 -9260.341} C_VEL
LIN {X 0,Y 439.307,Z 487.221,A -85,B 0,C 180,E1 -9261.722,E2 -9261.722} C_VEL
LIN {X 0,Y 438.965,Z 493.267,A -85,B 0,C 180,E1 -9263.272,E2 -9263.272} C_VEL
LIN {X 0,Y 438.22,Z 495.609,A -85,B 0,C 180,E1 -9263.975,E2 -9263.975} C_VEL
LIN {X 0,Y 435.195,Z 498.94,A -85,B 0,C 180,E1 -9265.134,E2 -9265.134} C_VEL
LIN {X 0,Y 432.658,Z 501.12,A -85,B 0,C 180,E1 -9266.09,E2 -9266.09} C_VEL
LIN {X 0,Y 431.56,Z 502.429,A -85,B 0,C 180,E1 -9266.843,E2 -9266.843} C_VEL
LIN {X 0,Y 431.466,Z 502.778,A -85,B 0,C 180,E1 -9267.099,E2 -9267.099} C_VEL
LIN {X 0,Y 431.384,Z 503.918,A -85,B 0,C 180,E1 -9268.133,E2 -9268.133} C_VEL
LIN {X 0,Y 431.282,Z 504.764,A -85,B 0,C 180,E1 -9270,E2 -9270} C_VEL
LIN {X 0,Y 431.312,Z 504.577,A -85,B 0,C 180,E1 -9270.934,E2 -9270.934} C_VEL
LIN {X 0,Y 431.453,Z 503.034,A -85,B 0,C 180,E1 -9272.801,E2 -9272.801} C_VEL
LIN {X 0,Y 431.543,Z 501.687,A -85,B 0,C 180,E1 -9273.735,E2 -9273.735} C_VEL
LIN {X 0,Y 431.553,Z 498.851,A -85,B 0,C 180,E1 -9275.139,E2 -9275.139} C_VEL
LIN {X 0,Y 431.875,Z 494.986,A -85,B 0,C 180,E1 -9276.541,E2 -9276.541} C_VEL
LIN {X 0,Y 432.119,Z 490.009,A -85,B 0,C 180,E1 -9277.946,E2 -9277.946} C_VEL
LIN {X 0,Y 432.588,Z 483.732,A -85,B 0,C 180,E1 -9279.35,E2 -9279.35} C_VEL
LIN {X 0,Y 433.129,Z 475.871,A -85,B 0,C 180,E1 -9280.755,E2 -9280.755} C_VEL
LIN {X 0,Y 433.769,Z 466.089,A -85,B 0,C 180,E1 -9282.159,E2 -9282.159} C_VEL
LIN {X 0,Y 434.517,Z 455.913,A -85,B 0,C 180,E1 -9283.315,E2 -9283.315} C_VEL
LIN {X 0,Y 435.05,Z 444.894,A -85,B 0,C 180,E1 -9284.324,E2 -9284.324} C_VEL
LIN {X 0,Y 435.604,Z 434.478,A -85,B 0,C 180,E1 -9285.08,E2 -9285.08} C_VEL
LIN {X 0,Y 436.134,Z 421.919,A -85,B 0,C 180,E1 -9285.779,E2 -9285.779} C_VEL
LIN {X 0,Y 435.166,Z 416.066,A -85,B 0,C 180,E1 -9286.08,E2 -9286.08} C_VEL
LIN {X 0,Y 431.829,Z 403.146,A -85,B 0,C 180,E1 -9286.648,E2 -9286.648} C_VEL
LIN {X 0,Y 431.558,Z 401.738,A -85,B 0,C 180,E1 -9286.701,E2 -9286.701} C_VEL
LIN {X 0,Y 431.536,Z 398.12,A -85,B 0,C 180,E1 -9289.999,E2 -9289.999} C_VEL
LIN {X 0,Y 431.6,Z 394.997,A -85,B 0,C 180,E1 -9293.005,E2 -9293.005} C_VEL
LIN {X 0,Y 431.711,Z 391.981,A -85,B 0,C 180,E1 -9296.075,E2 -9296.075} C_VEL
LIN {X 0,Y 431.782,Z 388.953,A -85,B 0,C 180,E1 -9299.229,E2 -9299.229} C_VEL
LIN {X 0,Y 431.856,Z 386.96,A -85,B 0,C 180,E1 -9301.384,E2 -9301.384} C_VEL
LIN {X 0,Y 432.122,Z 386.658,A -85,B 0,C 180,E1 -9303.956,E2 -9303.956} C_VEL
LIN {X 0,Y 432.299,Z 386.636,A -85,B 0,C 180,E1 -9306.979,E2 -9306.979} C_VEL
LIN {X 0,Y 432.337,Z 386.632,A -85,B 0,C 180,E1 -9310.179,E2 -9310.179} C_VEL
LIN {X 0,Y 432.32,Z 386.632,A -85,B 0,C 180,E1 -9313.061,E2 -9313.061} C_VEL
LIN {X 0,Y 432.336,Z 386.63,A -85,B 0,C 180,E1 -9315.665,E2 -9315.665} C_VEL
LIN {X 0,Y 432.336,Z 386.633,A -85,B 0,C 180,E1 -9318.398,E2 -9318.398} C_VEL
LIN {X 0,Y 432.351,Z 386.629,A -85,B 0,C 180,E1 -9321.851,E2 -9321.851} C_VEL
LIN {X 0,Y 432.345,Z 386.628,A -85,B 0,C 180,E1 -9325.323,E2 -9325.323} C_VEL
LIN {X 0,Y 432.326,Z 386.633,A -85,B 0,C 180,E1 -9328.654,E2 -9328.654} C_VEL
LIN {X 0,Y 432.386,Z 386.626,A -85,B 0,C 180,E1 -9331.877,E2 -9331.877} C_VEL
LIN {X 0,Y 432.351,Z 386.627,A -85,B 0,C 180,E1 -9334.999,E2 -9334.999} C_VEL
LIN {X 0,Y 432.362,Z 386.631,A -85,B 0,C 180,E1 -9338.046,E2 -9338.046} C_VEL
LIN {X 0,Y 432.389,Z 386.623,A -85,B 0,C 180,E1 -9341.03,E2 -9341.03} C_VEL
LIN {X 0,Y 432.435,Z 386.62,A -85,B 0,C 180,E1 -9343.961,E2 -9343.961} C_VEL
LIN {X 0,Y 432.464,Z 386.617,A -85,B 0,C 180,E1 -9347.803,E2 -9347.803} C_VEL
LIN {X 0,Y 432.469,Z 386.617,A -85,B 0,C 180,E1 -9351.59,E2 -9351.59} C_VEL
LIN {X 0,Y 432.601,Z 386.598,A -85,B 0,C 180,E1 -9354.406,E2 -9354.406} C_VEL
LIN {X 0,Y 432.608,Z 386.599,A -85,B 0,C 180,E1 -9358.138,E2 -9358.138} C_VEL
LIN {X 0,Y 432.737,Z 386.583,A -85,B 0,C 180,E1 -9360,E2 -9360} C_VEL
LIN {X 0,Y 432.597,Z 386.596,A -85,B 0,C 180,E1 -9362.794,E2 -9362.794} C_VEL
LIN {X 0,Y 432.578,Z 386.599,A -85,B 0,C 180,E1 -9366.53,E2 -9366.53} C_VEL
LIN {X 0,Y 432.449,Z 386.619,A -85,B 0,C 180,E1 -9369.353,E2 -9369.353} C_VEL
LIN {X 0,Y 432.45,Z 386.616,A -85,B 0,C 180,E1 -9372.812,E2 -9372.812} C_VEL
LIN {X 0,Y 432.416,Z 386.618,A -85,B 0,C 180,E1 -9376.478,E2 -9376.478} C_VEL
LIN {X 0,Y 432.343,Z 386.63,A -85,B 0,C 180,E1 -9379.96,E2 -9379.96} C_VEL
LIN {X 0,Y 432.322,Z 386.635,A -85,B 0,C 180,E1 -9382.964,E2 -9382.964} C_VEL
LIN {X 0,Y 432.365,Z 386.626,A -85,B 0,C 180,E1 -9386.032,E2 -9386.032} C_VEL
LIN {X 0,Y 432.347,Z 386.633,A -85,B 0,C 180,E1 -9389.187,E2 -9389.187} C_VEL
LIN {X 0,Y 432.327,Z 386.631,A -85,B 0,C 180,E1 -9392.443,E2 -9392.443} C_VEL
LIN {X 0,Y 432.348,Z 386.631,A -85,B 0,C 180,E1 -9395.632,E2 -9395.632} C_VEL
LIN {X 0,Y 432.354,Z 386.631,A -85,B 0,C 180,E1 -9399.342,E2 -9399.342} C_VEL
LIN {X 0,Y 432.337,Z 386.634,A -85,B 0,C 180,E1 -9401.797,E2 -9401.797} C_VEL
LIN {X 0,Y 432.337,Z 386.633,A -85,B 0,C 180,E1 -9404.347,E2 -9404.347} C_VEL
LIN {X 0,Y 432.375,Z 386.765,A -85,B 0,C 180,E1 -9407.894,E2 -9407.894} C_VEL
LIN {X 0,Y 433.419,Z 392.592,A -85,B 0,C 180,E1 -9410.773,E2 -9410.773} C_VEL
LIN {X 0,Y 434.332,Z 397.852,A -85,B 0,C 180,E1 -9413.222,E2 -9413.222} C_VEL
LIN {X 0,Y 434.349,Z 401.796,A -85,B 0,C 180,E1 -9414.941,E2 -9414.941} C_VEL
LIN {X 0,Y 433.833,Z 409.765,A -85,B 0,C 180,E1 -9418.231,E2 -9418.231} C_VEL
LIN {X 0,Y 433.289,Z 419.164,A -85,B 0,C 180,E1 -9421.94,E2 -9421.94} C_VEL
LIN {X 0,Y 432.779,Z 428.237,A -85,B 0,C 180,E1 -9425.422,E2 -9425.422} C_VEL
LIN {X 0,Y 432.321,Z 437.817,A -85,B 0,C 180,E1 -9429.044,E2 -9429.044} C_VEL
LIN {X 0,Y 431.997,Z 445.659,A -85,B 0,C 180,E1 -9431.995,E2 -9431.995} C_VEL
LIN {X 0,Y 431.869,Z 449.396,A -85,B 0,C 180,E1 -9433.304,E2 -9433.304} C_VEL
LIN {X 0,Y 434.063,Z 462.796,A -85,B 0,C 180,E1 -9433.763,E2 -9433.763} C_VEL
LIN {X 0,Y 435.639,Z 473.306,A -85,B 0,C 180,E1 -9434.262,E2 -9434.262} C_VEL
LIN {X 0,Y 435.091,Z 484.991,A -85,B 0,C 180,E1 -9434.902,E2 -9434.902} C_VEL
LIN {X 0,Y 434.425,Z 496.391,A -85,B 0,C 180,E1 -9435.717,E2 -9435.717} C_VEL
LIN {X 0,Y 433.804,Z 507.422,A -85,B 0,C 180,E1 -9436.714,E2 -9436.714} C_VEL
LIN {X 0,Y 433.231,Z 517.346,A -85,B 0,C 180,E1 -9437.825,E2 -9437.825} C_VEL
LIN {X 0,Y 432.576,Z 525.871,A -85,B 0,C 180,E1 -9438.994,E2 -9438.994} C_VEL
LIN {X 0,Y 432.103,Z 534.204,A -85,B 0,C 180,E1 -9440.403,E2 -9440.403} C_VEL
LIN {X 0,Y 431.711,Z 540.924,A -85,B 0,C 180,E1 -9441.811,E2 -9441.811} C_VEL
LIN {X 0,Y 431.459,Z 547.316,A -85,B 0,C 180,E1 -9443.528,E2 -9443.528} C_VEL
LIN {X 0,Y 431.369,Z 551.089,A -85,B 0,C 180,E1 -9444.859,E2 -9444.859} C_VEL
LIN {X 0,Y 431.21,Z 554.042,A -85,B 0,C 180,E1 -9446.262,E2 -9446.262} C_VEL
LIN {X 0,Y 431.28,Z 555.457,A -85,B 0,C 180,E1 -9447.198,E2 -9447.198} C_VEL
LIN {X 0,Y 431.198,Z 557.073,A -85,B 0,C 180,E1 -9449.066,E2 -9449.066} C_VEL
LIN {X 0,Y 431.216,Z 557.293,A -85,B 0,C 180,E1 -9450,E2 -9450} C_VEL
LIN {X 0,Y 431.198,Z 557.074,A -85,B 0,C 180,E1 -9450.934,E2 -9450.934} C_VEL
LIN {X 0,Y 431.28,Z 555.461,A -85,B 0,C 180,E1 -9452.802,E2 -9452.802} C_VEL
LIN {X 0,Y 431.21,Z 554.046,A -85,B 0,C 180,E1 -9453.738,E2 -9453.738} C_VEL
LIN {X 0,Y 431.369,Z 551.09,A -85,B 0,C 180,E1 -9455.141,E2 -9455.141} C_VEL
LIN {X 0,Y 431.441,Z 547.08,A -85,B 0,C 180,E1 -9456.547,E2 -9456.547} C_VEL
LIN {X 0,Y 431.712,Z 540.925,A -85,B 0,C 180,E1 -9458.189,E2 -9458.189} C_VEL
LIN {X 0,Y 432.103,Z 534.206,A -85,B 0,C 180,E1 -9459.597,E2 -9459.597} C_VEL
LIN {X 0,Y 432.574,Z 525.873,A -85,B 0,C 180,E1 -9461.005,E2 -9461.005} C_VEL
LIN {X 0,Y 433.221,Z 517.348,A -85,B 0,C 180,E1 -9462.175,E2 -9462.175} C_VEL
LIN {X 0,Y 433.806,Z 507.413,A -85,B 0,C 180,E1 -9463.287,E2 -9463.287} C_VEL
LIN {X 0,Y 434.412,Z 496.396,A -85,B 0,C 180,E1 -9464.283,E2 -9464.283} C_VEL
LIN {X 0,Y 435.076,Z 484.991,A -85,B 0,C 180,E1 -9465.098,E2 -9465.098} C_VEL
LIN {X 0,Y 435.607,Z 473.298,A -85,B 0,C 180,E1 -9465.739,E2 -9465.739} C_VEL
LIN {X 0,Y 433.58,Z 459.876,A -85,B 0,C 180,E1 -9466.351,E2 -9466.351} C_VEL
LIN {X 0,Y 431.871,Z 449.041,A -85,B 0,C 180,E1 -9466.721,E2 -9466.721} C_VEL
LIN {X 0,Y 432.209,Z 440.441,A -85,B 0,C 180,E1 -9469.967,E2 -9469.967} C_VEL
LIN {X 0,Y 432.556,Z 432.528,A -85,B 0,C 180,E1 -9472.951,E2 -9472.951} C_VEL
LIN {X 0,Y 433.03,Z 423.42,A -85,B 0,C 180,E1 -9476.396,E2 -9476.396} C_VEL
LIN {X 0,Y 433.36,Z 416.394,A -85,B 0,C 180,E1 -9479.112,E2 -9479.112} C_VEL
LIN {X 0,Y 433.896,Z 408.381,A -85,B 0,C 180,E1 -9482.311,E2 -9482.311} C_VEL
LIN {X 0,Y 434.35,Z 401.767,A -85,B 0,C 180,E1 -9485.058,E2 -9485.058} C_VEL
LIN {X 0,Y 434.285,Z 397.807,A -85,B 0,C 180,E1 -9486.782,E2 -9486.782} C_VEL
LIN {X 0,Y 433.236,Z 391.455,A -85,B 0,C 180,E1 -9489.758,E2 -9489.758} C_VEL
LIN {X 0,Y 432.375,Z 386.632,A -85,B 0,C 180,E1 -9492.262,E2 -9492.262} C_VEL
LIN {X 0,Y 432.335,Z 386.641,A -85,B 0,C 180,E1 -9495.665,E2 -9495.665} C_VEL
LIN {X 0,Y 432.335,Z 386.629,A -85,B 0,C 180,E1 -9498.398,E2 -9498.398} C_VEL
LIN {X 0,Y 432.35,Z 386.628,A -85,B 0,C 180,E1 -9501.851,E2 -9501.851} C_VEL
LIN {X 0,Y 432.343,Z 386.631,A -85,B 0,C 180,E1 -9505.323,E2 -9505.323} C_VEL
LIN {X 0,Y 432.324,Z 386.634,A -85,B 0,C 180,E1 -9508.654,E2 -9508.654} C_VEL
LIN {X 0,Y 432.385,Z 386.622,A -85,B 0,C 180,E1 -9511.877,E2 -9511.877} C_VEL
LIN {X 0,Y 432.349,Z 386.63,A -85,B 0,C 180,E1 -9514.999,E2 -9514.999} C_VEL
LIN {X 0,Y 432.36,Z 386.628,A -85,B 0,C 180,E1 -9518.046,E2 -9518.046} C_VEL
LIN {X 0,Y 432.39,Z 386.625,A -85,B 0,C 180,E1 -9521.03,E2 -9521.03} C_VEL
LIN {X 0,Y 432.434,Z 386.617,A -85,B 0,C 180,E1 -9523.961,E2 -9523.961} C_VEL
LIN {X 0,Y 432.484,Z 386.612,A -85,B 0,C 180,E1 -9527.804,E2 -9527.804} C_VEL
LIN {X 0,Y 432.496,Z 386.61,A -85,B 0,C 180,E1 -9531.59,E2 -9531.59} C_VEL
LIN {X 0,Y 432.601,Z 386.6,A -85,B 0,C 180,E1 -9534.406,E2 -9534.406} C_VEL
LIN {X 0,Y 432.608,Z 386.599,A -85,B 0,C 180,E1 -9538.138,E2 -9538.138} C_VEL
LIN {X 0,Y 432.738,Z 386.582,A -85,B 0,C 180,E1 -9540,E2 -9540} C_VEL
LIN {X 0,Y 432.595,Z 386.6,A -85,B 0,C 180,E1 -9542.794,E2 -9542.794} C_VEL
LIN {X 0,Y 432.577,Z 386.604,A -85,B 0,C 180,E1 -9546.53,E2 -9546.53} C_VEL
LIN {X 0,Y 432.445,Z 386.615,A -85,B 0,C 180,E1 -9549.353,E2 -9549.353} C_VEL
LIN {X 0,Y 432.434,Z 386.618,A -85,B 0,C 180,E1 -9552.804,E2 -9552.804} C_VEL
LIN {X 0,Y 432.415,Z 386.623,A -85,B 0,C 180,E1 -9556.479,E2 -9556.479} C_VEL
LIN {X 0,Y 432.342,Z 386.632,A -85,B 0,C 180,E1 -9559.96,E2 -9559.96} C_VEL
LIN {X 0,Y 432.321,Z 386.63,A -85,B 0,C 180,E1 -9562.964,E2 -9562.964} C_VEL
LIN {X 0,Y 432.364,Z 386.629,A -85,B 0,C 180,E1 -9566.033,E2 -9566.033} C_VEL
LIN {X 0,Y 432.346,Z 386.629,A -85,B 0,C 180,E1 -9569.187,E2 -9569.187} C_VEL
LIN {X 0,Y 432.326,Z 386.632,A -85,B 0,C 180,E1 -9572.443,E2 -9572.443} C_VEL
LIN {X 0,Y 432.347,Z 386.631,A -85,B 0,C 180,E1 -9575.632,E2 -9575.632} C_VEL
LIN {X 0,Y 432.355,Z 386.627,A -85,B 0,C 180,E1 -9578.717,E2 -9578.717} C_VEL
LIN {X 0,Y 432.336,Z 386.633,A -85,B 0,C 180,E1 -9581.797,E2 -9581.797} C_VEL
LIN {X 0,Y 432.381,Z 386.627,A -85,B 0,C 180,E1 -9585.659,E2 -9585.659} C_VEL
LIN {X 0,Y 432.371,Z 386.624,A -85,B 0,C 180,E1 -9588.393,E2 -9588.393} C_VEL
LIN {X 0,Y 432.337,Z 386.632,A -85,B 0,C 180,E1 -9591.85,E2 -9591.85} C_VEL
LIN {X 0,Y 432.195,Z 386.652,A -85,B 0,C 180,E1 -9595.309,E2 -9595.309} C_VEL
LIN {X 0,Y 431.831,Z 386.865,A -85,B 0,C 180,E1 -9598.614,E2 -9598.614} C_VEL
LIN {X 0,Y 431.768,Z 389.913,A -85,B 0,C 180,E1 -9601.833,E2 -9601.833} C_VEL
LIN {X 0,Y 431.668,Z 392.867,A -85,B 0,C 180,E1 -9604.956,E2 -9604.956} C_VEL
LIN {X 0,Y 431.585,Z 396.068,A -85,B 0,C 180,E1 -9608.156,E2 -9608.156} C_VEL
LIN {X 0,Y 431.596,Z 399.061,A -85,B 0,C 180,E1 -9610.993,E2 -9610.993} C_VEL
LIN {X 0,Y 431.565,Z 402.006,A -85,B 0,C 180,E1 -9613.404,E2 -9613.404} C_VEL
LIN {X 0,Y 434.954,Z 415.388,A -85,B 0,C 180,E1 -9613.978,E2 -9613.978} C_VEL
LIN {X 0,Y 436.143,Z 421.186,A -85,B 0,C 180,E1 -9614.281,E2 -9614.281} C_VEL
LIN {X 0,Y 435.698,Z 433.078,A -85,B 0,C 180,E1 -9614.924,E2 -9614.924} C_VEL
LIN {X 0,Y 435.176,Z 443.954,A -85,B 0,C 180,E1 -9615.695,E2 -9615.695} C_VEL
LIN {X 0,Y 434.564,Z 454.895,A -85,B 0,C 180,E1 -9616.676,E2 -9616.676} C_VEL
LIN {X 0,Y 433.8,Z 465.359,A -85,B 0,C 180,E1 -9617.842,E2 -9617.842} C_VEL
LIN {X 0,Y 433.26,Z 473.82,A -85,B 0,C 180,E1 -9619.012,E2 -9619.012} C_VEL
LIN {X 0,Y 432.712,Z 482.034,A -85,B 0,C 180,E1 -9620.417,E2 -9620.417} C_VEL
LIN {X 0,Y 432.288,Z 487.655,A -85,B 0,C 180,E1 -9621.586,E2 -9621.586} C_VEL
LIN {X 0,Y 431.927,Z 493.901,A -85,B 0,C 180,E1 -9623.221,E2 -9623.221} C_VEL
LIN {X 0,Y 431.556,Z 498.64,A -85,B 0,C 180,E1 -9624.861,E2 -9624.861} C_VEL
LIN {X 0,Y 431.543,Z 501.534,A -85,B 0,C 180,E1 -9626.265,E2 -9626.265} C_VEL
LIN {X 0,Y 431.466,Z 502.778,A -85,B 0,C 180,E1 -9627.099,E2 -9627.099} C_VEL
LIN {X 0,Y 430.764,Z 503.804,A -85,B 0,C 180,E1 -9627.866,E2 -9627.866} C_VEL
LIN {X 0,Y 427.822,Z 504.906,A -85,B 0,C 180,E1 -9629.122,E2 -9629.122} C_VEL
LIN {X 0,Y 425.358,Z 505.182,A -85,B 0,C 180,E1 -9630.141,E2 -9630.141} C_VEL
LIN {X 0,Y 424.318,Z 505.012,A -85,B 0,C 180,E1 -9630.929,E2 -9630.929} C_VEL
LIN {X 0,Y 424.244,Z 504.856,A -85,B 0,C 180,E1 -9631.196,E2 -9631.196} C_VEL
LIN {X 0,Y 424.384,Z 503.464,A -85,B 0,C 180,E1 -9632.848,E2 -9632.848} C_VEL
LIN {X 0,Y 424.487,Z 502.117,A -85,B 0,C 180,E1 -9633.797,E2 -9633.797} C_VEL
LIN {X 0,Y 424.484,Z 499.283,A -85,B 0,C 180,E1 -9635.225,E2 -9635.225} C_VEL
LIN {X 0,Y 424.835,Z 495.416,A -85,B 0,C 180,E1 -9636.65,E2 -9636.65} C_VEL
LIN {X 0,Y 425.094,Z 490.439,A -85,B 0,C 180,E1 -9638.079,E2 -9638.079} C_VEL
LIN {X 0,Y 425.589,Z 484.161,A -85,B 0,C 180,E1 -9639.505,E2 -9639.505} C_VEL
LIN {X 0,Y 426.173,Z 476.3,A -85,B 0,C 180,E1 -9640.932,E2 -9640.932} C_VEL
LIN {X 0,Y 426.737,Z 468.282,A -85,B 0,C 180,E1 -9642.121,E2 -9642.121} C_VEL
LIN {X 0,Y 427.47,Z 458.487,A -85,B 0,C 180,E1 -9643.307,E2 -9643.307} C_VEL
LIN {X 0,Y 428.026,Z 448.85,A -85,B 0,C 180,E1 -9644.258,E2 -9644.258} C_VEL
LIN {X 0,Y 428.619,Z 438.413,A -85,B 0,C 180,E1 -9645.088,E2 -9645.088} C_VEL
LIN {X 0,Y 429.178,Z 425.833,A -85,B 0,C 180,E1 -9645.859,E2 -9645.859} C_VEL
LIN {X 0,Y 429.129,Z 421.059,A -85,B 0,C 180,E1 -9646.105,E2 -9646.105} C_VEL
LIN {X 0,Y 426.189,Z 408.623,A -85,B 0,C 180,E1 -9646.726,E2 -9646.726} C_VEL
LIN {X 0,Y 424.481,Z 402.153,A -85,B 0,C 180,E1 -9646.992,E2 -9646.992} C_VEL
LIN {X 0,Y 424.477,Z 398.506,A -85,B 0,C 180,E1 -9650.347,E2 -9650.347} C_VEL
LIN {X 0,Y 424.55,Z 395.356,A -85,B 0,C 180,E1 -9653.41,E2 -9653.41} C_VEL
LIN {X 0,Y 424.649,Z 392.314,A -85,B 0,C 180,E1 -9656.542,E2 -9656.542} C_VEL
LIN {X 0,Y 424.749,Z 389.254,A -85,B 0,C 180,E1 -9659.762,E2 -9659.762} C_VEL
LIN {X 0,Y 424.845,Z 387.566,A -85,B 0,C 180,E1 -9661.963,E2 -9661.963} C_VEL
LIN {X 0,Y 425.205,Z 387.518,A -85,B 0,C 180,E1 -9665.345,E2 -9665.345} C_VEL
LIN {X 0,Y 425.279,Z 387.509,A -85,B 0,C 180,E1 -9667.695,E2 -9667.695} C_VEL
LIN {X 0,Y 425.283,Z 387.513,A -85,B 0,C 180,E1 -9670.52,E2 -9670.52} C_VEL
LIN {X 0,Y 425.261,Z 387.51,A -85,B 0,C 180,E1 -9673.351,E2 -9673.351} C_VEL
LIN {X 0,Y 425.261,Z 387.514,A -85,B 0,C 180,E1 -9676.649,E2 -9676.649} C_VEL
LIN {X 0,Y 425.299,Z 387.509,A -85,B 0,C 180,E1 -9679.874,E2 -9679.874} C_VEL
LIN {X 0,Y 425.289,Z 387.511,A -85,B 0,C 180,E1 -9682.487,E2 -9682.487} C_VEL
LIN {X 0,Y 425.312,Z 387.506,A -85,B 0,C 180,E1 -9685.818,E2 -9685.818} C_VEL
LIN {X 0,Y 425.295,Z 387.507,A -85,B 0,C 180,E1 -9689.239,E2 -9689.239} C_VEL
LIN {X 0,Y 425.353,Z 387.503,A -85,B 0,C 180,E1 -9692.442,E2 -9692.442} C_VEL
LIN {X 0,Y 425.352,Z 387.501,A -85,B 0,C 180,E1 -9695.602,E2 -9695.602} C_VEL
LIN {X 0,Y 425.298,Z 387.506,A -85,B 0,C 180,E1 -9698.682,E2 -9698.682} C_VEL
LIN {X 0,Y 425.335,Z 387.506,A -85,B 0,C 180,E1 -9701.703,E2 -9701.703} C_VEL
LIN {X 0,Y 425.353,Z 387.5,A -85,B 0,C 180,E1 -9704.671,E2 -9704.671} C_VEL
LIN {X 0,Y 425.417,Z 387.494,A -85,B 0,C 180,E1 -9707.598,E2 -9707.598} C_VEL
LIN {X 0,Y 425.413,Z 387.494,A -85,B 0,C 180,E1 -9711.449,E2 -9711.449} C_VEL
LIN {X 0,Y 425.556,Z 387.476,A -85,B 0,C 180,E1 -9714.313,E2 -9714.313} C_VEL
LIN {X 0,Y 425.578,Z 387.474,A -85,B 0,C 180,E1 -9718.107,E2 -9718.107} C_VEL
LIN {X 0,Y 425.707,Z 387.458,A -85,B 0,C 180,E1 -9720,E2 -9720} C_VEL
LIN {X 0,Y 425.55,Z 387.473,A -85,B 0,C 180,E1 -9722.84,E2 -9722.84} C_VEL
LIN {X 0,Y 425.536,Z 387.476,A -85,B 0,C 180,E1 -9726.639,E2 -9726.639} C_VEL
LIN {X 0,Y 425.408,Z 387.496,A -85,B 0,C 180,E1 -9729.509,E2 -9729.509} C_VEL
LIN {X 0,Y 425.409,Z 387.494,A -85,B 0,C 180,E1 -9732.91,E2 -9732.91} C_VEL
LIN {X 0,Y 425.365,Z 387.497,A -85,B 0,C 180,E1 -9736.605,E2 -9736.605} C_VEL
LIN {X 0,Y 425.333,Z 387.505,A -85,B 0,C 180,E1 -9739.636,E2 -9739.636} C_VEL
LIN {X 0,Y 425.309,Z 387.508,A -85,B 0,C 180,E1 -9743.365,E2 -9743.365} C_VEL
LIN {X 0,Y 425.352,Z 387.501,A -85,B 0,C 180,E1 -9746.844,E2 -9746.844} C_VEL
LIN {X 0,Y 425.295,Z 387.507,A -85,B 0,C 180,E1 -9749.719,E2 -9749.719} C_VEL
LIN {X 0,Y 425.286,Z 387.512,A -85,B 0,C 180,E1 -9753.048,E2 -9753.048} C_VEL
LIN {X 0,Y 425.287,Z 387.508,A -85,B 0,C 180,E1 -9755.929,E2 -9755.929} C_VEL
LIN {X 0,Y 425.301,Z 387.509,A -85,B 0,C 180,E1 -9759.043,E2 -9759.043} C_VEL
LIN {X 0,Y 425.278,Z 387.514,A -85,B 0,C 180,E1 -9762.653,E2 -9762.653} C_VEL
LIN {X 0,Y 425.272,Z 387.513,A -85,B 0,C 180,E1 -9766.045,E2 -9766.045} C_VEL
LIN {X 0,Y 425.35,Z 387.663,A -85,B 0,C 180,E1 -9767.56,E2 -9767.56} C_VEL
LIN {X 0,Y 426.491,Z 394.033,A -85,B 0,C 180,E1 -9770.76,E2 -9770.76} C_VEL
LIN {X 0,Y 427.322,Z 398.962,A -85,B 0,C 180,E1 -9773.109,E2 -9773.109} C_VEL
LIN {X 0,Y 427.38,Z 402.902,A -85,B 0,C 180,E1 -9774.861,E2 -9774.861} C_VEL
LIN {X 0,Y 426.836,Z 410.859,A -85,B 0,C 180,E1 -9778.204,E2 -9778.204} C_VEL
LIN {X 0,Y 426.245,Z 420.223,A -85,B 0,C 180,E1 -9781.971,E2 -9781.971} C_VEL
LIN {X 0,Y 425.696,Z 429.57,A -85,B 0,C 180,E1 -9785.623,E2 -9785.623} C_VEL
LIN {X 0,Y 425.237,Z 438.8,A -85,B 0,C 180,E1 -9789.186,E2 -9789.186} C_VEL
LIN {X 0,Y 424.896,Z 446.604,A -85,B 0,C 180,E1 -9792.181,E2 -9792.181} C_VEL
LIN {X 0,Y 424.79,Z 448.725,A -85,B 0,C 180,E1 -9792.993,E2 -9792.993} C_VEL
LIN {X 0,Y 427.268,Z 464.198,A -85,B 0,C 180,E1 -9793.569,E2 -9793.569} C_VEL
LIN {X 0,Y 428.678,Z 475.218,A -85,B 0,C 180,E1 -9794.122,E2 -9794.122} C_VEL
LIN {X 0,Y 427.98,Z 488.101,A -85,B 0,C 180,E1 -9794.889,E2 -9794.889} C_VEL
LIN {X 0,Y 427.342,Z 498.819,A -85,B 0,C 180,E1 -9795.718,E2 -9795.718} C_VEL
LIN {X 0,Y 426.754,Z 508.699,A -85,B 0,C 180,E1 -9796.67,E2 -9796.67} C_VEL
LIN {X 0,Y 426.113,Z 518.719,A -85,B 0,C 180,E1 -9797.861,E2 -9797.861} C_VEL
LIN {X 0,Y 425.387,Z 528.435,A -85,B 0,C 180,E1 -9799.288,E2 -9799.288} C_VEL
LIN {X 0,Y 424.902,Z 536.183,A -85,B 0,C 180,E1 -9800.719,E2 -9800.719} C_VEL
LIN {X 0,Y 424.465,Z 543.328,A -85,B 0,C 180,E1 -9802.388,E2 -9802.388} C_VEL
LIN {X 0,Y 424.289,Z 548.424,A -85,B 0,C 180,E1 -9803.929,E2 -9803.929} C_VEL
LIN {X 0,Y 424.226,Z 551.734,A -85,B 0,C 180,E1 -9805.248,E2 -9805.248} C_VEL
LIN {X 0,Y 424.121,Z 553.609,A -85,B 0,C 180,E1 -9806.199,E2 -9806.199} C_VEL
LIN {X 0,Y 424.192,Z 555.025,A -85,B 0,C 180,E1 -9807.151,E2 -9807.151} C_VEL
LIN {X 0,Y 424.115,Z 556.642,A -85,B 0,C 180,E1 -9809.05,E2 -9809.05} C_VEL
LIN {X 0,Y 424.13,Z 556.862,A -85,B 0,C 180,E1 -9810,E2 -9810} C_VEL
LIN {X 0,Y 424.115,Z 556.643,A -85,B 0,C 180,E1 -9810.949,E2 -9810.949} C_VEL
LIN {X 0,Y 424.192,Z 555.028,A -85,B 0,C 180,E1 -9812.849,E2 -9812.849} C_VEL
LIN {X 0,Y 424.121,Z 553.613,A -85,B 0,C 180,E1 -9813.8,E2 -9813.8} C_VEL
LIN {X 0,Y 424.279,Z 550.657,A -85,B 0,C 180,E1 -9815.227,E2 -9815.227} C_VEL
LIN {X 0,Y 424.359,Z 546.646,A -85,B 0,C 180,E1 -9816.657,E2 -9816.657} C_VEL
LIN {X 0,Y 424.651,Z 540.49,A -85,B 0,C 180,E1 -9818.326,E2 -9818.326} C_VEL
LIN {X 0,Y 425.047,Z 533.77,A -85,B 0,C 180,E1 -9819.758,E2 -9819.758} C_VEL
LIN {X 0,Y 425.566,Z 525.438,A -85,B 0,C 180,E1 -9821.189,E2 -9821.189} C_VEL
LIN {X 0,Y 426.238,Z 516.912,A -85,B 0,C 180,E1 -9822.377,E2 -9822.377} C_VEL
LIN {X 0,Y 426.878,Z 506.23,A -85,B 0,C 180,E1 -9823.583,E2 -9823.583} C_VEL
LIN {X 0,Y 427.581,Z 494.527,A -85,B 0,C 180,E1 -9824.638,E2 -9824.638} C_VEL
LIN {X 0,Y 428.361,Z 482.633,A -85,B 0,C 180,E1 -9825.463,E2 -9825.463} C_VEL
LIN {X 0,Y 428.687,Z 474.077,A -85,B 0,C 180,E1 -9825.938,E2 -9825.938} C_VEL
LIN {X 0,Y 426.789,Z 461.17,A -85,B 0,C 180,E1 -9826.561,E2 -9826.561} C_VEL
LIN {X 0,Y 424.79,Z 448.677,A -85,B 0,C 180,E1 -9827.008,E2 -9827.008} C_VEL
LIN {X 0,Y 425.108,Z 442.089,A -85,B 0,C 180,E1 -9829.551,E2 -9829.551} C_VEL
LIN {X 0,Y 425.468,Z 433.534,A -85,B 0,C 180,E1 -9832.841,E2 -9832.841} C_VEL
LIN {X 0,Y 425.903,Z 425.531,A -85,B 0,C 180,E1 -9835.931,E2 -9835.931} C_VEL
LIN {X 0,Y 426.347,Z 417.42,A -85,B 0,C 180,E1 -9839.113,E2 -9839.113} C_VEL
LIN {X 0,Y 426.882,Z 409.464,A -85,B 0,C 180,E1 -9842.348,E2 -9842.348} C_VEL
LIN {X 0,Y 427.38,Z 402.876,A -85,B 0,C 180,E1 -9845.139,E2 -9845.139} C_VEL
LIN {X 0,Y 427.29,Z 398.929,A -85,B 0,C 180,E1 -9846.894,E2 -9846.894} C_VEL
LIN {X 0,Y 426.225,Z 392.41,A -85,B 0,C 180,E1 -9850.021,E2 -9850.021} C_VEL
LIN {X 0,Y 425.333,Z 387.511,A -85,B 0,C 180,E1 -9852.553,E2 -9852.553} C_VEL
LIN {X 0,Y 425.263,Z 387.516,A -85,B 0,C 180,E1 -9856.044,E2 -9856.044} C_VEL
LIN {X 0,Y 425.277,Z 387.51,A -85,B 0,C 180,E1 -9858.622,E2 -9858.622} C_VEL
LIN {X 0,Y 425.318,Z 387.507,A -85,B 0,C 180,E1 -9861.103,E2 -9861.103} C_VEL
LIN {X 0,Y 425.303,Z 387.509,A -85,B 0,C 180,E1 -9864.664,E2 -9864.664} C_VEL
LIN {X 0,Y 425.268,Z 387.51,A -85,B 0,C 180,E1 -9868.073,E2 -9868.073} C_VEL
LIN {X 0,Y 425.334,Z 387.501,A -85,B 0,C 180,E1 -9871.368,E2 -9871.368} C_VEL
LIN {X 0,Y 425.357,Z 387.499,A -85,B 0,C 180,E1 -9873.506,E2 -9873.506} C_VEL
LIN {X 0,Y 425.308,Z 387.508,A -85,B 0,C 180,E1 -9876.635,E2 -9876.635} C_VEL
LIN {X 0,Y 425.332,Z 387.505,A -85,B 0,C 180,E1 -9880.364,E2 -9880.364} C_VEL
LIN {X 0,Y 425.392,Z 387.493,A -85,B 0,C 180,E1 -9883.688,E2 -9883.688} C_VEL
LIN {X 0,Y 425.434,Z 387.489,A -85,B 0,C 180,E1 -9887.599,E2 -9887.599} C_VEL
LIN {X 0,Y 425.446,Z 387.488,A -85,B 0,C 180,E1 -9891.45,E2 -9891.45} C_VEL
LIN {X 0,Y 425.557,Z 387.477,A -85,B 0,C 180,E1 -9894.313,E2 -9894.313} C_VEL
LIN {X 0,Y 425.577,Z 387.474,A -85,B 0,C 180,E1 -9898.107,E2 -9898.107} C_VEL
LIN {X 0,Y 425.707,Z 387.458,A -85,B 0,C 180,E1 -9900,E2 -9900} C_VEL
LIN {X 0,Y 425.548,Z 387.477,A -85,B 0,C 180,E1 -9902.84,E2 -9902.84} C_VEL
LIN {X 0,Y 425.534,Z 387.479,A -85,B 0,C 180,E1 -9906.648,E2 -9906.648} C_VEL
LIN {X 0,Y 425.403,Z 387.493,A -85,B 0,C 180,E1 -9909.509,E2 -9909.509} C_VEL
LIN {X 0,Y 425.397,Z 387.494,A -85,B 0,C 180,E1 -9912.904,E2 -9912.904} C_VEL
LIN {X 0,Y 425.364,Z 387.5,A -85,B 0,C 180,E1 -9916.605,E2 -9916.605} C_VEL
LIN {X 0,Y 425.332,Z 387.504,A -85,B 0,C 180,E1 -9919.636,E2 -9919.636} C_VEL
LIN {X 0,Y 425.291,Z 387.509,A -85,B 0,C 180,E1 -9922.339,E2 -9922.339} C_VEL
LIN {X 0,Y 425.294,Z 387.508,A -85,B 0,C 180,E1 -9925.446,E2 -9925.446} C_VEL
LIN {X 0,Y 425.352,Z 387.502,A -85,B 0,C 180,E1 -9927.558,E2 -9927.558} C_VEL
LIN {X 0,Y 425.291,Z 387.507,A -85,B 0,C 180,E1 -9930.816,E2 -9930.816} C_VEL
LIN {X 0,Y 425.314,Z 387.506,A -85,B 0,C 180,E1 -9934.288,E2 -9934.288} C_VEL
LIN {X 0,Y 425.288,Z 387.512,A -85,B 0,C 180,E1 -9937.694,E2 -9937.694} C_VEL
LIN {X 0,Y 425.287,Z 387.508,A -85,B 0,C 180,E1 -9940.521,E2 -9940.521} C_VEL
LIN {X 0,Y 425.26,Z 387.514,A -85,B 0,C 180,E1 -9943.351,E2 -9943.351} C_VEL
LIN {X 0,Y 425.319,Z 387.503,A -85,B 0,C 180,E1 -9946.641,E2 -9946.641} C_VEL
LIN {X 0,Y 425.285,Z 387.512,A -85,B 0,C 180,E1 -9949.479,E2 -9949.479} C_VEL
LIN {X 0,Y 425.275,Z 387.509,A -85,B 0,C 180,E1 -9952.489,E2 -9952.489} C_VEL
LIN {X 0,Y 425.121,Z 387.533,A -85,B 0,C 180,E1 -9955.75,E2 -9955.75} C_VEL
LIN {X 0,Y 424.84,Z 387.568,A -85,B 0,C 180,E1 -9958.037,E2 -9958.037} C_VEL
LIN {X 0,Y 424.759,Z 388.371,A -85,B 0,C 180,E1 -9959.36,E2 -9959.36} C_VEL
LIN {X 0,Y 424.677,Z 391.212,A -85,B 0,C 180,E1 -9962.395,E2 -9962.395} C_VEL
LIN {X 0,Y 424.636,Z 394.215,A -85,B 0,C 180,E1 -9965.558,E2 -9965.558} C_VEL
LIN {X 0,Y 424.518,Z 397.331,A -85,B 0,C 180,E1 -9968.641,E2 -9968.641} C_VEL
LIN {X 0,Y 424.479,Z 400.582,A -85,B 0,C 180,E1 -9971.665,E2 -9971.665} C_VEL
LIN {X 0,Y 424.46,Z 402.207,A -85,B 0,C 180,E1 -9973.107,E2 -9973.107} C_VEL
LIN {X 0,Y 428.109,Z 416.299,A -85,B 0,C 180,E1 -9973.734,E2 -9973.734} C_VEL
LIN {X 0,Y 429.299,Z 422.919,A -85,B 0,C 180,E1 -9974.085,E2 -9974.085} C_VEL
LIN {X 0,Y 428.752,Z 435.3,A -85,B 0,C 180,E1 -9974.795,E2 -9974.795} C_VEL
LIN {X 0,Y 428.189,Z 446.308,A -85,B 0,C 180,E1 -9975.62,E2 -9975.62} C_VEL
LIN {X 0,Y 427.489,Z 457.654,A -85,B 0,C 180,E1 -9976.693,E2 -9976.693} C_VEL
LIN {X 0,Y 426.771,Z 467.597,A -85,B 0,C 180,E1 -9977.88,E2 -9977.88} C_VEL
LIN {X 0,Y 426.083,Z 477.199,A -85,B 0,C 180,E1 -9979.306,E2 -9979.306} C_VEL
LIN {X 0,Y 425.521,Z 484.855,A -85,B 0,C 180,E1 -9980.733,E2 -9980.733} C_VEL
LIN {X 0,Y 425.008,Z 491.875,A -85,B 0,C 180,E1 -9982.398,E2 -9982.398} C_VEL
LIN {X 0,Y 424.725,Z 496.547,A -85,B 0,C 180,E1 -9983.826,E2 -9983.826} C_VEL
LIN {X 0,Y 424.509,Z 500.123,A -85,B 0,C 180,E1 -9985.252,E2 -9985.252} C_VEL
LIN {X 0,Y 424.487,Z 501.966,A -85,B 0,C 180,E1 -9986.203,E2 -9986.203} C_VEL
LIN {X 0,Y 424.393,Z 503.359,A -85,B 0,C 180,E1 -9987.152,E2 -9987.152} C_VEL
LIN {X 0,Y 424.239,Z 504.961,A -85,B 0,C 180,E1 -9989.051,E2 -9989.051} C_VEL
LIN {X 0,Y 424.224,Z 505.194,A -85,B 0,C 180,E1 -9990,E2 -9990} C_VEL
LIN {X 0,Y 424.244,Z 504.856,A -85,B 0,C 180,E1 -9991.196,E2 -9991.196} C_VEL
LIN {X 0,Y 423.602,Z 504.412,A -85,B 0,C 180,E1 -9991.989,E2 -9991.989} C_VEL
LIN {X 0,Y 420.773,Z 503.193,A -85,B 0,C 180,E1 -9993.274,E2 -9993.274} C_VEL
LIN {X 0,Y 417.988,Z 501.323,A -85,B 0,C 180,E1 -9994.556,E2 -9994.556} C_VEL
LIN {X 0,Y 417.426,Z 499.662,A -85,B 0,C 180,E1 -9995.334,E2 -9995.334} C_VEL
LIN {X 0,Y 417.795,Z 495.018,A -85,B 0,C 180,E1 -9997.03,E2 -9997.03} C_VEL
LIN {X 0,Y 418.238,Z 488.907,A -85,B 0,C 180,E1 -9998.699,E2 -9998.699} C_VEL
LIN {X 0,Y 418.802,Z 482.155,A -85,B 0,C 180,E1 -10000.149,E2 -10000.149} C_VEL
LIN {X 0,Y 419.46,Z 473.717,A -85,B 0,C 180,E1 -10001.599,E2 -10001.599} C_VEL
LIN {X 0,Y 420.147,Z 465.032,A -85,B 0,C 180,E1 -10002.806,E2 -10002.806} C_VEL
LIN {X 0,Y 420.868,Z 454.95,A -85,B 0,C 180,E1 -10003.947,E2 -10003.947} C_VEL
LIN {X 0,Y 421.439,Z 444.205,A -85,B 0,C 180,E1 -10004.931,E2 -10004.931} C_VEL
LIN {X 0,Y 422.065,Z 433.512,A -85,B 0,C 180,E1 -10005.699,E2 -10005.699} C_VEL
LIN {X 0,Y 422.409,Z 422.825,A -85,B 0,C 180,E1 -10006.303,E2 -10006.303} C_VEL
LIN {X 0,Y 419.469,Z 410.223,A -85,B 0,C 180,E1 -10006.961,E2 -10006.961} C_VEL
LIN {X 0,Y 417.424,Z 402.573,A -85,B 0,C 180,E1 -10007.286,E2 -10007.286} C_VEL
LIN {X 0,Y 417.416,Z 398.893,A -85,B 0,C 180,E1 -10010.706,E2 -10010.706} C_VEL
LIN {X 0,Y 417.504,Z 395.717,A -85,B 0,C 180,E1 -10013.829,E2 -10013.829} C_VEL
LIN {X 0,Y 417.59,Z 392.651,A -85,B 0,C 180,E1 -10017.027,E2 -10017.027} C_VEL
LIN {X 0,Y 417.714,Z 389.556,A -85,B 0,C 180,E1 -10020.315,E2 -10020.315} C_VEL
LIN {X 0,Y 417.75,Z 388.54,A -85,B 0,C 180,E1 -10021.435,E2 -10021.435} C_VEL
LIN {X 0,Y 418.116,Z 388.404,A -85,B 0,C 180,E1 -10024.855,E2 -10024.855} C_VEL
LIN {X 0,Y 418.228,Z 388.387,A -85,B 0,C 180,E1 -10027.833,E2 -10027.833} C_VEL
LIN {X 0,Y 418.225,Z 388.388,A -85,B 0,C 180,E1 -10030.948,E2 -10030.948} C_VEL
LIN {X 0,Y 418.213,Z 388.389,A -85,B 0,C 180,E1 -10033.729,E2 -10033.729} C_VEL
LIN {X 0,Y 418.212,Z 388.392,A -85,B 0,C 180,E1 -10036.449,E2 -10036.449} C_VEL
LIN {X 0,Y 418.228,Z 388.387,A -85,B 0,C 180,E1 -10039.13,E2 -10039.13} C_VEL
LIN {X 0,Y 418.239,Z 388.389,A -85,B 0,C 180,E1 -10042.165,E2 -10042.165} C_VEL
LIN {X 0,Y 418.27,Z 388.381,A -85,B 0,C 180,E1 -10045.42,E2 -10045.42} C_VEL
LIN {X 0,Y 418.216,Z 388.391,A -85,B 0,C 180,E1 -10048.604,E2 -10048.604} C_VEL
LIN {X 0,Y 418.295,Z 388.382,A -85,B 0,C 180,E1 -10051.937,E2 -10051.937} C_VEL
LIN {X 0,Y 418.294,Z 388.378,A -85,B 0,C 180,E1 -10055.163,E2 -10055.163} C_VEL
LIN {X 0,Y 418.239,Z 388.388,A -85,B 0,C 180,E1 -10058.304,E2 -10058.304} C_VEL
LIN {X 0,Y 418.286,Z 388.381,A -85,B 0,C 180,E1 -10061.383,E2 -10061.383} C_VEL
LIN {X 0,Y 418.307,Z 388.379,A -85,B 0,C 180,E1 -10064.406,E2 -10064.406} C_VEL
LIN {X 0,Y 418.36,Z 388.372,A -85,B 0,C 180,E1 -10067.386,E2 -10067.386} C_VEL
LIN {X 0,Y 418.344,Z 388.373,A -85,B 0,C 180,E1 -10070.329,E2 -10070.329} C_VEL
LIN {X 0,Y 418.484,Z 388.356,A -85,B 0,C 180,E1 -10073.249,E2 -10073.249} C_VEL
LIN {X 0,Y 418.342,Z 388.374,A -85,B 0,C 180,E1 -10075.182,E2 -10075.182} C_VEL
LIN {X 0,Y 418.547,Z 388.35,A -85,B 0,C 180,E1 -10078.075,E2 -10078.075} C_VEL
LIN {X 0,Y 418.676,Z 388.334,A -85,B 0,C 180,E1 -10080,E2 -10080} C_VEL
LIN {X 0,Y 418.505,Z 388.351,A -85,B 0,C 180,E1 -10082.888,E2 -10082.888} C_VEL
LIN {X 0,Y 418.499,Z 388.353,A -85,B 0,C 180,E1 -10086.751,E2 -10086.751} C_VEL
LIN {X 0,Y 418.364,Z 388.374,A -85,B 0,C 180,E1 -10089.671,E2 -10089.671} C_VEL
LIN {X 0,Y 418.36,Z 388.372,A -85,B 0,C 180,E1 -10093.006,E2 -10093.006} C_VEL
LIN {X 0,Y 418.317,Z 388.375,A -85,B 0,C 180,E1 -10096.735,E2 -10096.735} C_VEL
LIN {X 0,Y 418.275,Z 388.384,A -85,B 0,C 180,E1 -10099.79,E2 -10099.79} C_VEL
LIN {X 0,Y 418.242,Z 388.386,A -85,B 0,C 180,E1 -10102.736,E2 -10102.736} C_VEL
LIN {X 0,Y 418.273,Z 388.382,A -85,B 0,C 180,E1 -10105.904,E2 -10105.904} C_VEL
LIN {X 0,Y 418.269,Z 388.386,A -85,B 0,C 180,E1 -10109.162,E2 -10109.162} C_VEL
LIN {X 0,Y 418.261,Z 388.386,A -85,B 0,C 180,E1 -10112.844,E2 -10112.844} C_VEL
LIN {X 0,Y 418.25,Z 388.384,A -85,B 0,C 180,E1 -10116.238,E2 -10116.238} C_VEL
LIN {X 0,Y 418.255,Z 388.384,A -85,B 0,C 180,E1 -10119.682,E2 -10119.682} C_VEL
LIN {X 0,Y 418.233,Z 388.392,A -85,B 0,C 180,E1 -10122.321,E2 -10122.321} C_VEL
LIN {X 0,Y 418.243,Z 388.388,A -85,B 0,C 180,E1 -10125.109,E2 -10125.109} C_VEL
LIN {X 0,Y 418.275,Z 388.503,A -85,B 0,C 180,E1 -10127.176,E2 -10127.176} C_VEL
LIN {X 0,Y 419.221,Z 393.527,A -85,B 0,C 180,E1 -10129.802,E2 -10129.802} C_VEL
LIN {X 0,Y 420.317,Z 400.055,A -85,B 0,C 180,E1 -10132.99,E2 -10132.99} C_VEL
LIN {X 0,Y 420.381,Z 404.506,A -85,B 0,C 180,E1 -10135.004,E2 -10135.004} C_VEL
LIN {X 0,Y 419.82,Z 411.94,A -85,B 0,C 180,E1 -10138.175,E2 -10138.175} C_VEL
LIN {X 0,Y 419.209,Z 421.264,A -85,B 0,C 180,E1 -10142.003,E2 -10142.003} C_VEL
LIN {X 0,Y 418.674,Z 429.253,A -85,B 0,C 180,E1 -10145.187,E2 -10145.187} C_VEL
LIN {X 0,Y 418.287,Z 437.15,A -85,B 0,C 180,E1 -10148.306,E2 -10148.306} C_VEL
LIN {X 0,Y 417.93,Z 444.94,A -85,B 0,C 180,E1 -10151.367,E2 -10151.367} C_VEL
LIN {X 0,Y 417.736,Z 448.374,A -85,B 0,C 180,E1 -10152.713,E2 -10152.713} C_VEL
LIN {X 0,Y 419.975,Z 462.206,A -85,B 0,C 180,E1 -10153.214,E2 -10153.214} C_VEL
LIN {X 0,Y 421.757,Z 474.781,A -85,B 0,C 180,E1 -10153.854,E2 -10153.854} C_VEL
LIN {X 0,Y 421.244,Z 485.897,A -85,B 0,C 180,E1 -10154.517,E2 -10154.517} C_VEL
LIN {X 0,Y 420.435,Z 498.385,A -85,B 0,C 180,E1 -10155.478,E2 -10155.478} C_VEL
LIN {X 0,Y 419.732,Z 509.342,A -85,B 0,C 180,E1 -10156.566,E2 -10156.566} C_VEL
LIN {X 0,Y 419.139,Z 518.284,A -85,B 0,C 180,E1 -10157.655,E2 -10157.655} C_VEL
LIN {X 0,Y 418.45,Z 526.501,A -85,B 0,C 180,E1 -10158.863,E2 -10158.863} C_VEL
LIN {X 0,Y 417.928,Z 534.577,A -85,B 0,C 180,E1 -10160.319,E2 -10160.319} C_VEL
LIN {X 0,Y 417.539,Z 541.06,A -85,B 0,C 180,E1 -10161.774,E2 -10161.774} C_VEL
LIN {X 0,Y 417.259,Z 547.299,A -85,B 0,C 180,E1 -10163.594,E2 -10163.594} C_VEL
LIN {X 0,Y 417.162,Z 551.302,A -85,B 0,C 180,E1 -10165.168,E2 -10165.168} C_VEL
LIN {X 0,Y 417.036,Z 553.177,A -85,B 0,C 180,E1 -10166.135,E2 -10166.135} C_VEL
LIN {X 0,Y 417.107,Z 554.593,A -85,B 0,C 180,E1 -10167.102,E2 -10167.102} C_VEL
LIN {X 0,Y 417.035,Z 556.211,A -85,B 0,C 180,E1 -10169.034,E2 -10169.034} C_VEL
LIN {X 0,Y 417.047,Z 556.43,A -85,B 0,C 180,E1 -10170,E2 -10170} C_VEL
LIN {X 0,Y 417.035,Z 556.212,A -85,B 0,C 180,E1 -10170.966,E2 -10170.966} C_VEL
LIN {X 0,Y 417.107,Z 554.596,A -85,B 0,C 180,E1 -10172.897,E2 -10172.897} C_VEL
LIN {X 0,Y 417.036,Z 553.181,A -85,B 0,C 180,E1 -10173.865,E2 -10173.865} C_VEL
LIN {X 0,Y 417.192,Z 550.223,A -85,B 0,C 180,E1 -10175.316,E2 -10175.316} C_VEL
LIN {X 0,Y 417.276,Z 546.212,A -85,B 0,C 180,E1 -10176.771,E2 -10176.771} C_VEL
LIN {X 0,Y 417.588,Z 540.055,A -85,B 0,C 180,E1 -10178.468,E2 -10178.468} C_VEL
LIN {X 0,Y 418.015,Z 533.335,A -85,B 0,C 180,E1 -10179.923,E2 -10179.923} C_VEL
LIN {X 0,Y 418.573,Z 525.004,A -85,B 0,C 180,E1 -10181.378,E2 -10181.378} C_VEL
LIN {X 0,Y 419.239,Z 516.476,A -85,B 0,C 180,E1 -10182.587,E2 -10182.587} C_VEL
LIN {X 0,Y 419.92,Z 505.629,A -85,B 0,C 180,E1 -10183.83,E2 -10183.83} C_VEL
LIN {X 0,Y 420.702,Z 494.093,A -85,B 0,C 180,E1 -10184.883,E2 -10184.883} C_VEL
LIN {X 0,Y 421.517,Z 482.199,A -85,B 0,C 180,E1 -10185.72,E2 -10185.72} C_VEL
LIN {X 0,Y 421.767,Z 474.775,A -85,B 0,C 180,E1 -10186.145,E2 -10186.145} C_VEL
LIN {X 0,Y 419.893,Z 461.727,A -85,B 0,C 180,E1 -10186.807,E2 -10186.807} C_VEL
LIN {X 0,Y 417.736,Z 448.323,A -85,B 0,C 180,E1 -10187.287,E2 -10187.287} C_VEL
LIN {X 0,Y 418.062,Z 441.063,A -85,B 0,C 180,E1 -10190.158,E2 -10190.158} C_VEL
LIN {X 0,Y 418.479,Z 433.206,A -85,B 0,C 180,E1 -10193.245,E2 -10193.245} C_VEL
LIN {X 0,Y 418.931,Z 425.23,A -85,B 0,C 180,E1 -10196.396,E2 -10196.396} C_VEL
LIN {X 0,Y 419.357,Z 417.807,A -85,B 0,C 180,E1 -10199.37,E2 -10199.37} C_VEL
LIN {X 0,Y 419.867,Z 410.533,A -85,B 0,C 180,E1 -10202.387,E2 -10202.387} C_VEL
LIN {X 0,Y 420.377,Z 404.484,A -85,B 0,C 180,E1 -10204.995,E2 -10204.995} C_VEL
LIN {X 0,Y 420.298,Z 400.034,A -85,B 0,C 180,E1 -10207.011,E2 -10207.011} C_VEL
LIN {X 0,Y 419.225,Z 393.521,A -85,B 0,C 180,E1 -10210.197,E2 -10210.197} C_VEL
LIN {X 0,Y 418.266,Z 388.391,A -85,B 0,C 180,E1 -10212.906,E2 -10212.906} C_VEL
LIN {X 0,Y 418.212,Z 388.392,A -85,B 0,C 180,E1 -10216.271,E2 -10216.271} C_VEL
LIN {X 0,Y 418.227,Z 388.39,A -85,B 0,C 180,E1 -10219.13,E2 -10219.13} C_VEL
LIN {X 0,Y 418.237,Z 388.386,A -85,B 0,C 180,E1 -10222.165,E2 -10222.165} C_VEL
LIN {X 0,Y 418.268,Z 388.383,A -85,B 0,C 180,E1 -10225.42,E2 -10225.42} C_VEL
LIN {X 0,Y 418.214,Z 388.391,A -85,B 0,C 180,E1 -10228.604,E2 -10228.604} C_VEL
LIN {X 0,Y 418.294,Z 388.377,A -85,B 0,C 180,E1 -10231.937,E2 -10231.937} C_VEL
LIN {X 0,Y 418.292,Z 388.381,A -85,B 0,C 180,E1 -10235.163,E2 -10235.163} C_VEL
LIN {X 0,Y 418.237,Z 388.389,A -85,B 0,C 180,E1 -10238.304,E2 -10238.304} C_VEL
LIN {X 0,Y 418.287,Z 388.379,A -85,B 0,C 180,E1 -10241.383,E2 -10241.383} C_VEL
LIN {X 0,Y 418.306,Z 388.38,A -85,B 0,C 180,E1 -10244.406,E2 -10244.406} C_VEL
LIN {X 0,Y 418.374,Z 388.368,A -85,B 0,C 180,E1 -10247.386,E2 -10247.386} C_VEL
LIN {X 0,Y 418.363,Z 388.374,A -85,B 0,C 180,E1 -10250.329,E2 -10250.329} C_VEL
LIN {X 0,Y 418.497,Z 388.353,A -85,B 0,C 180,E1 -10253.249,E2 -10253.249} C_VEL
LIN {X 0,Y 418.341,Z 388.372,A -85,B 0,C 180,E1 -10255.182,E2 -10255.182} C_VEL
LIN {X 0,Y 418.546,Z 388.349,A -85,B 0,C 180,E1 -10258.076,E2 -10258.076} C_VEL
LIN {X 0,Y 418.677,Z 388.333,A -85,B 0,C 180,E1 -10260,E2 -10260} C_VEL
LIN {X 0,Y 418.504,Z 388.354,A -85,B 0,C 180,E1 -10262.888,E2 -10262.888} C_VEL
LIN {X 0,Y 418.498,Z 388.355,A -85,B 0,C 180,E1 -10266.751,E2 -10266.751} C_VEL
LIN {X 0,Y 418.403,Z 388.366,A -85,B 0,C 180,E1 -10268.695,E2 -10268.695} C_VEL
LIN {X 0,Y 418.359,Z 388.372,A -85,B 0,C 180,E1 -10272.614,E2 -10272.614} C_VEL
LIN {X 0,Y 418.305,Z 388.379,A -85,B 0,C 180,E1 -10275.594,E2 -10275.594} C_VEL
LIN {X 0,Y 418.285,Z 388.381,A -85,B 0,C 180,E1 -10278.617,E2 -10278.617} C_VEL
LIN {X 0,Y 418.237,Z 388.388,A -85,B 0,C 180,E1 -10281.696,E2 -10281.696} C_VEL
LIN {X 0,Y 418.287,Z 388.379,A -85,B 0,C 180,E1 -10284.864,E2 -10284.864} C_VEL
LIN {X 0,Y 418.295,Z 388.382,A -85,B 0,C 180,E1 -10288.063,E2 -10288.063} C_VEL
LIN {X 0,Y 418.215,Z 388.39,A -85,B 0,C 180,E1 -10291.396,E2 -10291.396} C_VEL
LIN {X 0,Y 418.268,Z 388.381,A -85,B 0,C 180,E1 -10294.58,E2 -10294.58} C_VEL
LIN {X 0,Y 418.238,Z 388.39,A -85,B 0,C 180,E1 -10297.835,E2 -10297.835} C_VEL
LIN {X 0,Y 418.226,Z 388.387,A -85,B 0,C 180,E1 -10300.948,E2 -10300.948} C_VEL
LIN {X 0,Y 418.212,Z 388.392,A -85,B 0,C 180,E1 -10303.729,E2 -10303.729} C_VEL
LIN {X 0,Y 418.275,Z 388.381,A -85,B 0,C 180,E1 -10306.457,E2 -10306.457} C_VEL
LIN {X 0,Y 418.263,Z 388.383,A -85,B 0,C 180,E1 -10309.124,E2 -10309.124} C_VEL
LIN {X 0,Y 418.227,Z 388.388,A -85,B 0,C 180,E1 -10312.167,E2 -10312.167} C_VEL
LIN {X 0,Y 418.116,Z 388.404,A -85,B 0,C 180,E1 -10315.145,E2 -10315.145} C_VEL
LIN {X 0,Y 417.879,Z 388.436,A -85,B 0,C 180,E1 -10317.44,E2 -10317.44} C_VEL
LIN {X 0,Y 417.706,Z 388.457,A -85,B 0,C 180,E1 -10318.561,E2 -10318.561} C_VEL
LIN {X 0,Y 417.645,Z 391.533,A -85,B 0,C 180,E1 -10321.889,E2 -10321.889} C_VEL
LIN {X 0,Y 417.571,Z 394.79,A -85,B 0,C 180,E1 -10325.348,E2 -10325.348} C_VEL
LIN {X 0,Y 417.474,Z 397.707,A -85,B 0,C 180,E1 -10328.262,E2 -10328.262} C_VEL
LIN {X 0,Y 417.447,Z 400.985,A -85,B 0,C 180,E1 -10331.344,E2 -10331.344} C_VEL
LIN {X 0,Y 417.418,Z 402.626,A -85,B 0,C 180,E1 -10332.816,E2 -10332.816} C_VEL
LIN {X 0,Y 420.893,Z 415.927,A -85,B 0,C 180,E1 -10333.412,E2 -10333.412} C_VEL
LIN {X 0,Y 422.461,Z 423.2,A -85,B 0,C 180,E1 -10333.812,E2 -10333.812} C_VEL
LIN {X 0,Y 421.934,Z 435.738,A -85,B 0,C 180,E1 -10334.544,E2 -10334.544} C_VEL
LIN {X 0,Y 421.233,Z 448.229,A -85,B 0,C 180,E1 -10335.507,E2 -10335.507} C_VEL
LIN {X 0,Y 420.618,Z 458.089,A -85,B 0,C 180,E1 -10336.472,E2 -10336.472} C_VEL
LIN {X 0,Y 419.852,Z 468.032,A -85,B 0,C 180,E1 -10337.677,E2 -10337.677} C_VEL
LIN {X 0,Y 419.137,Z 477.632,A -85,B 0,C 180,E1 -10339.127,E2 -10339.127} C_VEL
LIN {X 0,Y 418.529,Z 485.289,A -85,B 0,C 180,E1 -10340.577,E2 -10340.577} C_VEL
LIN {X 0,Y 417.989,Z 492.308,A -85,B 0,C 180,E1 -10342.27,E2 -10342.27} C_VEL
LIN {X 0,Y 417.697,Z 496.979,A -85,B 0,C 180,E1 -10343.721,E2 -10343.721} C_VEL
LIN {X 0,Y 417.429,Z 500.557,A -85,B 0,C 180,E1 -10345.171,E2 -10345.171} C_VEL
LIN {X 0,Y 417.431,Z 502.397,A -85,B 0,C 180,E1 -10346.139,E2 -10346.139} C_VEL
LIN {X 0,Y 417.325,Z 503.79,A -85,B 0,C 180,E1 -10347.104,E2 -10347.104} C_VEL
LIN {X 0,Y 417.154,Z 505.393,A -85,B 0,C 180,E1 -10349.035,E2 -10349.035} C_VEL
LIN {X 0,Y 417.15,Z 505.625,A -85,B 0,C 180,E1 -10350,E2 -10350} C_VEL
LIN {X 0,Y 417.223,Z 504.856,A -85,B 0,C 180,E1 -10351.931,E2 -10351.931} C_VEL
LIN {X 0,Y 417.431,Z 502.547,A -85,B 0,C 180,E1 -10353.862,E2 -10353.862} C_VEL
LIN {X 0,Y 417.426,Z 499.662,A -85,B 0,C 180,E1 -10355.334,E2 -10355.334} C_VEL
LIN {X 0,Y 416.893,Z 497.826,A -85,B 0,C 180,E1 -10356.1,E2 -10356.1} C_VEL
LIN {X 0,Y 414.284,Z 494.428,A -85,B 0,C 180,E1 -10357.339,E2 -10357.339} C_VEL
LIN {X 0,Y 411.775,Z 490.461,A -85,B 0,C 180,E1 -10358.552,E2 -10358.552} C_VEL
LIN {X 0,Y 411.398,Z 487.566,A -85,B 0,C 180,E1 -10359.267,E2 -10359.267} C_VEL
LIN {X 0,Y 412.019,Z 479.964,A -85,B 0,C 180,E1 -10360.815,E2 -10360.815} C_VEL
LIN {X 0,Y 412.774,Z 470.901,A -85,B 0,C 180,E1 -10362.288,E2 -10362.288} C_VEL
LIN {X 0,Y 413.536,Z 461.464,A -85,B 0,C 180,E1 -10363.514,E2 -10363.514} C_VEL
LIN {X 0,Y 414.245,Z 450.846,A -85,B 0,C 180,E1 -10364.631,E2 -10364.631} C_VEL
LIN {X 0,Y 414.974,Z 439.261,A -85,B 0,C 180,E1 -10365.596,E2 -10365.596} C_VEL
LIN {X 0,Y 415.539,Z 427.477,A -85,B 0,C 180,E1 -10366.349,E2 -10366.349} C_VEL
LIN {X 0,Y 415.652,Z 424.317,A -85,B 0,C 180,E1 -10366.522,E2 -10366.522} C_VEL
LIN {X 0,Y 412.734,Z 411.802,A -85,B 0,C 180,E1 -10367.206,E2 -10367.206} C_VEL
LIN {X 0,Y 410.368,Z 402.983,A -85,B 0,C 180,E1 -10367.603,E2 -10367.603} C_VEL
LIN {X 0,Y 410.37,Z 399.281,A -85,B 0,C 180,E1 -10371.079,E2 -10371.079} C_VEL
LIN {X 0,Y 410.53,Z 395.483,A -85,B 0,C 180,E1 -10374.861,E2 -10374.861} C_VEL
LIN {X 0,Y 410.603,Z 391.939,A -85,B 0,C 180,E1 -10378.637,E2 -10378.637} C_VEL
LIN {X 0,Y 410.732,Z 389.592,A -85,B 0,C 180,E1 -10381.179,E2 -10381.179} C_VEL
LIN {X 0,Y 410.856,Z 389.31,A -85,B 0,C 180,E1 -10383.188,E2 -10383.188} C_VEL
LIN {X 0,Y 411.093,Z 389.275,A -85,B 0,C 180,E1 -10385.54,E2 -10385.54} C_VEL
LIN {X 0,Y 411.206,Z 389.264,A -85,B 0,C 180,E1 -10388.168,E2 -10388.168} C_VEL
LIN {X 0,Y 411.167,Z 389.265,A -85,B 0,C 180,E1 -10391.228,E2 -10391.228} C_VEL
LIN {X 0,Y 411.179,Z 389.268,A -85,B 0,C 180,E1 -10394.491,E2 -10394.491} C_VEL
LIN {X 0,Y 411.181,Z 389.268,A -85,B 0,C 180,E1 -10398.195,E2 -10398.195} C_VEL
LIN {X 0,Y 411.228,Z 389.26,A -85,B 0,C 180,E1 -10400.777,E2 -10400.777} C_VEL
LIN {X 0,Y 411.204,Z 389.265,A -85,B 0,C 180,E1 -10404.472,E2 -10404.472} C_VEL
LIN {X 0,Y 411.211,Z 389.261,A -85,B 0,C 180,E1 -10406.873,E2 -10406.873} C_VEL
LIN {X 0,Y 411.237,Z 389.259,A -85,B 0,C 180,E1 -10410.644,E2 -10410.644} C_VEL
LIN {X 0,Y 411.241,Z 389.259,A -85,B 0,C 180,E1 -10413.619,E2 -10413.619} C_VEL
LIN {X 0,Y 411.2,Z 389.261,A -85,B 0,C 180,E1 -10416.852,E2 -10416.852} C_VEL
LIN {X 0,Y 411.22,Z 389.264,A -85,B 0,C 180,E1 -10420.05,E2 -10420.05} C_VEL
LIN {X 0,Y 411.267,Z 389.254,A -85,B 0,C 180,E1 -10423.131,E2 -10423.131} C_VEL
LIN {X 0,Y 411.31,Z 389.248,A -85,B 0,C 180,E1 -10426.896,E2 -10426.896} C_VEL
LIN {X 0,Y 411.296,Z 389.252,A -85,B 0,C 180,E1 -10430.161,E2 -10430.161} C_VEL
LIN {X 0,Y 411.447,Z 389.232,A -85,B 0,C 180,E1 -10433.133,E2 -10433.133} C_VEL
LIN {X 0,Y 411.313,Z 389.249,A -85,B 0,C 180,E1 -10435.099,E2 -10435.099} C_VEL
LIN {X 0,Y 411.516,Z 389.226,A -85,B 0,C 180,E1 -10438.043,E2 -10438.043} C_VEL
LIN {X 0,Y 411.645,Z 389.21,A -85,B 0,C 180,E1 -10440,E2 -10440} C_VEL
LIN {X 0,Y 411.462,Z 389.229,A -85,B 0,C 180,E1 -10442.937,E2 -10442.937} C_VEL
LIN {X 0,Y 411.466,Z 389.229,A -85,B 0,C 180,E1 -10446.867,E2 -10446.867} C_VEL
LIN {X 0,Y 411.313,Z 389.252,A -85,B 0,C 180,E1 -10449.838,E2 -10449.838} C_VEL
LIN {X 0,Y 411.318,Z 389.25,A -85,B 0,C 180,E1 -10453.109,E2 -10453.109} C_VEL
LIN {X 0,Y 411.261,Z 389.255,A -85,B 0,C 180,E1 -10456.889,E2 -10456.889} C_VEL
LIN {X 0,Y 411.235,Z 389.259,A -85,B 0,C 180,E1 -10459.987,E2 -10459.987} C_VEL
LIN {X 0,Y 411.206,Z 389.265,A -85,B 0,C 180,E1 -10463.147,E2 -10463.147} C_VEL
LIN {X 0,Y 411.241,Z 389.257,A -85,B 0,C 180,E1 -10466.381,E2 -10466.381} C_VEL
LIN {X 0,Y 411.204,Z 389.263,A -85,B 0,C 180,E1 -10469.712,E2 -10469.712} C_VEL
LIN {X 0,Y 411.21,Z 389.265,A -85,B 0,C 180,E1 -10473.156,E2 -10473.156} C_VEL
LIN {X 0,Y 411.197,Z 389.264,A -85,B 0,C 180,E1 -10476.553,E2 -10476.553} C_VEL
LIN {X 0,Y 411.218,Z 389.26,A -85,B 0,C 180,E1 -10479.728,E2 -10479.728} C_VEL
LIN {X 0,Y 411.177,Z 389.27,A -85,B 0,C 180,E1 -10483.133,E2 -10483.133} C_VEL
LIN {X 0,Y 411.204,Z 389.339,A -85,B 0,C 180,E1 -10486.786,E2 -10486.786} C_VEL
LIN {X 0,Y 412.365,Z 395.51,A -85,B 0,C 180,E1 -10490.08,E2 -10490.08} C_VEL
LIN {X 0,Y 413.375,Z 401.514,A -85,B 0,C 180,E1 -10493.042,E2 -10493.042} C_VEL
LIN {X 0,Y 413.434,Z 405.084,A -85,B 0,C 180,E1 -10494.692,E2 -10494.692} C_VEL
LIN {X 0,Y 412.747,Z 413.525,A -85,B 0,C 180,E1 -10498.361,E2 -10498.361} C_VEL
LIN {X 0,Y 412.163,Z 422.296,A -85,B 0,C 180,E1 -10502.036,E2 -10502.036} C_VEL
LIN {X 0,Y 411.608,Z 430.323,A -85,B 0,C 180,E1 -10505.302,E2 -10505.302} C_VEL
LIN {X 0,Y 411.191,Z 438.1,A -85,B 0,C 180,E1 -10508.44,E2 -10508.44} C_VEL
LIN {X 0,Y 410.815,Z 445.831,A -85,B 0,C 180,E1 -10511.549,E2 -10511.549} C_VEL
